# B&R Automation Studio project NAEUL004C00R13L518F00 (part 63)

#### InputRef_Link.var - Change By Project
```iecst
(*2019-06-28*)
(**)
VAR
	p_bLinkStartupRun : REFERENCE TO BOOL;
	p_eLinkMcParamUSCommMod : REFERENCE TO eMcSetCommMod;
	p_bLinkNtParamProjLaneBPrep : REFERENCE TO BOOL;
	bHermesRun : BOOL;
	bHermesStop : BOOL;
END_VAR
(**)
VAR
	p_bLinkDILeftSen : REFERENCE TO BOOL;
	p_eLinkTravLifULPosGo : REFERENCE TO eTravLifULPos;
	p_bLinkOpsTravLifULUSComm : REFERENCE TO BOOL;
END_VAR
(**)
VAR
	sWidthInUMTemp : STRING[80];
END_VAR
```

#### Act_LinkAction.st - Change By Project
```iecst
(** 2021-08-01 **)
ACTION Act_LinkAction:

	IF p_bLinkStartupRun = TRUE THEN
		p_eAct ACCESS p_StartupUSHermesBAct;
	ELSE
		p_eAct ACCESS ADR(eAct);

		IF EDGEPOS(p_eLinkMcParamUSCommMod = McSetCommModHermes AND p_bLinkNtParamProjLaneBPrep) THEN
			bHermesRun	:= TRUE;
			bHermesStop	:= FALSE;
		END_IF

		IF EDGENEG(p_eLinkMcParamUSCommMod = McSetCommModHermes AND p_bLinkNtParamProjLaneBPrep) THEN
			bHermesRun	:= FALSE;
			bHermesStop	:= TRUE;
		END_IF

		IF bHermesRun = TRUE THEN
			p_eAct	:= HermesActBGStartRun;

			IF (eStat = HermesActBGStartRun) AND (eStatus = Done) THEN
				p_eAct		:= HermesActIdle;
				bHermesRun	:= FALSE;
			END_IF
		END_IF

		IF bHermesStop = TRUE THEN
			p_eAct	:= HermesActBGStopRun;

			IF (eStat = HermesActBGStopRun) AND (eStatus = Done) THEN
				p_eAct		:= HermesActIdle;
				bHermesStop	:= FALSE;
			END_IF
		END_IF

		fbDlyTmr(IN := TRUE);
		IF fbDlyTmr.Q THEN
			fbDeleteLogTmr (IN := TRUE);
			IF fbDeleteLogTmr.Q AND eStatus <> Busy THEN
				p_eAct := HermesActDeleteOldLog;
				IF eStat = HermesActDeleteOldLog AND eStatus = Done THEN
					p_eAct := HermesActIdle;
					fbDlyTmr (IN := FALSE);
					fbDeleteLogTmr (IN := FALSE);
				END_IF
			END_IF
		END_IF

	END_IF

END_ACTION
```

#### Act_Link.st - Change By Project
```iecst
(** 2019-06-04 **)
ACTION Act_Link:

	//Receive Alive Time
	p_tyParam.tRcvAlive	:= p_tyParam.tSndAlive * 2;

	//Transfer Complete
	p_bRcvCompl	:= EDGENEG(p_bLinkDILeftSen);

	//Ready Receive
	p_bRdyRcv	:= p_bLinkOpsTravLifULUSComm AND p_eLinkTravLifULPosGo = TravLifULPosUS2;

	//Ready Transport
	p_bRdyTransport	:= TRUE;

	//Accept Data Ready
	IF bUSRdy AND p_eLinkTravLifULPosGo = TravLifULPosUS2 THEN
		p_bAccDataRdy	:= TRUE;
	ELSIF bUSRdy = FALSE THEN
		p_bAccDataRdy	:= FALSE;
	END_IF

	//Accept New Recipe Condition
	p_bAccNewRcpCond	:= p_bOpsRun = TRUE;

	//Info Message
	p_sInfoMsg		:= 'Upstream Hermes Request New Recipe';
	p_sInfoMsg		:= CONCAT(p_sInfoMsg , '$r$n');
	p_sInfoMsg		:= CONCAT(p_sInfoMsg , 'Old Recipe Name : ');
	p_sInfoMsg		:= CONCAT(p_sInfoMsg , p_sRecipeNm);
	p_sInfoMsg		:= CONCAT(p_sInfoMsg , '$r$n');
	p_sInfoMsg		:= CONCAT(p_sInfoMsg , 'Old Recipe Width : ');
	sWidthInUMTemp	:= DINT_TO_STRING(p_diWidthInUM / 1000);
	p_sInfoMsg		:= CONCAT(p_sInfoMsg , sWidthInUMTemp);
	p_sInfoMsg		:= CONCAT(p_sInfoMsg , '$r$n');
	p_sInfoMsg		:= CONCAT(p_sInfoMsg , 'New Recipe Name : ');
	p_sInfoMsg		:= CONCAT(p_sInfoMsg , sReqRecipeNm);
	p_sInfoMsg		:= CONCAT(p_sInfoMsg , '$r$n');
	p_sInfoMsg		:= CONCAT(p_sInfoMsg , 'New Recipe Width : ');
	sWidthInUMTemp	:= DINT_TO_STRING(diReqWidthInUM / 1000);
	p_sInfoMsg		:= CONCAT(p_sInfoMsg , sWidthInUMTemp);

	//Info Message 1 for "SendBoardInfo"
	p_sInfoMsg1     := 'Board Info Received From Upstream';
	p_sInfoMsg1		:= CONCAT(p_sInfoMsg1 , '$r$n');
	p_sInfoMsg1		:= CONCAT(p_sInfoMsg1 , 'PCB Transfer to Last Zone is Blocked');
	p_sInfoMsg1		:= CONCAT(p_sInfoMsg1 , '$r$n');
	p_sInfoMsg1		:= CONCAT(p_sInfoMsg1 , 'Please Insert PCB to Last Zone Outlet');
	p_sInfoMsg1		:= CONCAT(p_sInfoMsg1 , '$r$n');
	p_sInfoMsg1		:= CONCAT(p_sInfoMsg1 , 'and PCB Data Will Be Overwritten');
	p_sInfoMsg1		:= CONCAT(p_sInfoMsg1 , '$r$n');
	p_sInfoMsg1		:= CONCAT(p_sInfoMsg1 , 'To Cancel,unpress the Query Board Info Button');

	//Info Message 2 for "SendBoardInfo"
	p_sInfoMsg2     := 'Board Info Not Found From Upstream';

	//Block Upstream
	//ADD
	//Changed
	bBlkUS :=  bBABlkUS OR bBFBlkUS OR bManuallInsertLastZone; // OR (p_eLinkMcParamUSCommMod = McSetCommModHermes AND (p_bQueryBypassWorkOrder OR p_bNewIncomingBoard)) ; //Remove bManuallInsertLastZone if this is a multiple zones, use bManuallInsertLastZone to block respective zones board transfer

	//Changed
	//For first machine ?
//	IF p_bNewIncomingBoard = FALSE THEN
//		fbUSBlkTm(IN := TRUE);
//	ELSIF p_bNewIncomingBoard THEN
//		fbUSBlkTm(IN := FALSE);
//	END_IF

	//IF AutoRcp Prep, Link
	IF p_bNtParamAutoRcpPrep AND NOT(p_bMcParamAutoRcpDis) AND p_eNtParamAutoRcpPrecededBy = PrecededBySelf   THEN
		p_sRecipeNm	ACCESS p_AutoRcpCurrRcpProdID;
		p_diWidthInUM ACCESS p_AutoRcpCurrRcpWidth;
	ELSE
		p_sRecipeNm	ACCESS p_ProdRcpCurrRcp0Nm;
		p_diWidthInUM ACCESS p_ProdRcpCurrRcp0Width;
	END_IF

END_ACTION
```

#### Cyclic.st - Do Not Change!!!
```iecst
(** 2021-08-01 **)
PROGRAM _CYCLIC

	IF bInitDone = FALSE THEN
		bInitDone	:= TRUE;

		Act_InitLocal;
		Act_InitGlobal;

	ELSIF bInitialDone = FALSE THEN
		IF p_bNtSettingsLoadDone = TRUE THEN
			bInitialDone	:= TRUE;

			Act_Initial;
		END_IF

	ELSE

		Act_RstErr;
		Act_LinkAction;
		Act_Action;
		Act_LinkEn;

		IF (p_bPrep = TRUE) AND (p_bEn = TRUE) AND (p_bDis = FALSE) THEN
			Act_Link;
			Act_Main;
			Act_Background;
			Act_Background_ProcessData;
		ELSE
			Act_Main_Disable;

			IF eStat <> HermesActIdle THEN
				eStatus	:= Done;
			ELSE
				eStatus	:= Idle;
			END_IF
		END_IF

		Act_CombineErr;
		Act_Alarm;
		Act_Alarm1;
		Act_Alarm2;
		Act_Alarm3;
		Act_Alarm4;
		Act_Alarm5;
	END_IF

END_PROGRAM
```

#### Act_InitLocal.st - Do Not Change!!!
```iecst
(** 2021-08-01 **)
ACTION Act_InitLocal:

	//Input Reference Link To Local Variable
	p_eAct ACCESS ADR(eAct);
	p_udiRstErr ACCESS ADR(udiRstErr);
	p_bPrep ACCESS ADR(bPrep);
	p_bEn ACCESS ADR(bEn);
	p_bDis ACCESS ADR(bDis);
	p_tyParam ACCESS ADR(tyParam);
	p_sIPAddr ACCESS ADR(sIPAddr);
	p_tyDTStructure ACCESS ADR(tyDTStructure);
	p_dtCurrDT ACCESS ADR(dtCurrDT);
	p_bRdyRcv ACCESS ADR(bRdyRcv);
	p_bRdyTransport ACCESS ADR(bRdyTransport);
	p_bRcvCompl ACCESS ADR(bRcvCompl);
	p_bRcvIncompl ACCESS ADR(bRcvInCompl);
	p_bRcvNotStart ACCESS ADR(bRcvNotStart);
	p_bBAWidthEn ACCESS ADR(bBAWidthEn);
	p_bBASltEn ACCESS ADR(bBASltEn);
	p_bBFWidthEn ACCESS ADR(bBFWidthEn);
	p_bBFSltEn ACCESS ADR(bBFSltEn);
	p_sMcId ACCESS ADR(sMcId);
	p_sInterfaceId ACCESS ADR(sInterfaceId);
	p_sVersion ACCESS ADR(sVersion);
	p_eFailedBoard ACCESS ADR(eFailedBoard);
	p_sRecipeNm ACCESS ADR(sRecipeNm);
	p_diWidthInUM ACCESS ADR(diWidthInUM);
	p_diMinSltValue ACCESS ADR(diMinSltValue);
	p_diMaxSltValue ACCESS ADR(diMaxSltValue);
	p_diPitch ACCESS ADR(diPitch);
	p_diTtlSlt ACCESS ADR(diTtlSlt);
	p_diSltToSltInUM ACCESS ADR(diSltToSltInUM);
	p_udiSndBffrSize ACCESS ADR(udiSndBffrSize);
	p_udiRcvBffrSize ACCESS ADR(udiRcvBffrSize);
	p_udiAliveIdleTimeInSec ACCESS ADR(udiAliveIdleTimeInSec);
	p_tConnTimeOut ACCESS ADR(tConnTimeOut);
	p_diTransferInTO ACCESS ADR(diTransferInTO);
	p_bOpsRun ACCESS ADR(bOpsRun);
	p_bInterruptSen ACCESS ADR(bInterruptSen);
	p_udiFileKeepDay ACCESS ADR(udiFileKeepDay);
	p_sProgNm ACCESS ADR(sProgNm);
	p_bNtSettingsLoadDone ACCESS ADR(bNtSettingsLoadDone);
	p_bAccDataRdy ACCESS ADR(bAccDataRdy);
	p_bRmtPrep ACCESS ADR(bRmtPrep);
	p_bRmtEn ACCESS ADR(bRmtEn);
	p_bSvyPrep ACCESS ADR(bSvyPrep);
	p_bSvyEn ACCESS ADR(bSvyEn);
	pa_tyProdRcpList ACCESS ADR(a_tyProdRcpList);
	p_tyProdRcpCurrRcp ACCESS ADR(tyProdRcpCurrRcp);
	p_bMcParamMnlAccData ACCESS ADR(bMcParamMnlAccData);
	p_bOpsGConv1HvBrd ACCESS ADR(bOpsGConv1HvBrd);
	p_bManualInsertEndSen ACCESS ADR(bManualInsertEndSen);
	p_bManualInsertZoneHvBrd ACCESS ADR(bManualInsertZoneHvBrd);
	p_bUIAccData ACCESS ADR(bUIAccData);
    p_bQueryBoardInfo ACCESS ADR(bQueryBoardInfo);
	p_sTopBarcode ACCESS ADR(sTopBarcode);
	p_sBottomBarcode ACCESS ADR(sBottomBarcode);
	p_tyHermesConfiguration ACCESS ADR(tyHermesCurrConfiguration);
	p_bTransportFinished ACCESS ADR(bTransportFinished);
	p_bInternalUse ACCESS ADR(bInternalUse);
	p_sInternalRcv ACCESS ADR(sInternalRcv);
	p_bAccNewRcpCond ACCESS ADR(bAccNewRcpCond);
	p_sInfoMsg ACCESS ADR(sInfoMsg);
	p_sInfoMsg1 ACCESS ADR(sInfoMsg1);
	p_sInfoMsg2 ACCESS ADR(sInfoMsg2);

END_ACTION
```

#### Act_Initial.st - Do Not Change!!!
```iecst
(** 2021-08-01 **)
ACTION Act_Initial:

	//Initial
	sStatTxt	:= a_sStatText[eStat];

	fbClntConnect.udiSndBffrSize		:= p_udiSndBffrSize;
	fbClntConnect.udiRcvBffrSize		:= p_udiRcvBffrSize;
	fbClntConnect.udiAliveIdleTmInSec	:= p_udiAliveIdleTimeInSec;
	fbClntConnect.tConnectTO			:= p_tConnTimeOut;
	fbClntConnect(bEn := FALSE);

	fbRcv.udiBffrSize	:= SIZEOF(sRcv);
	fbRcv.p_BffrDest	:= ADR(sRcv);
	fbRcv(bEn := FALSE);

	fbSend.p_BffrDest	:= ADR(sSnd);
	fbSend(bEn := FALSE);

	fbClose(bEn := FALSE);

	fbParseXMLTable.p_XMLTable	:= ADR(a_tyXMLTableDataRcv);

	fbCheckAlive(bEn := FALSE);

	fbCheckAliveSendPing(bEn := FALSE);

	fbCheckAliveRcvPing(bEn := FALSE);

	fbSequenceUS.p_tyMsgTypeRcv	:= ADR(tyMsgTypeRcv);
	fbSequenceUS(bEn := FALSE);

	fbSequenceTO(bEn := FALSE);

	fbFileAppend1.sDevice	:= 'Log';
	fbFileAppend1(bEn := FALSE);

	fbFileOldDel1.sDevice			:= 'Log';
	fbFileOldDel1.sPath				:= '';
	fbFileOldDel1.sKeyword			:= p_sProgNm;
	fbFileOldDel1.udiFileKeepDay	:= p_udiFileKeepDay;
	fbFileOldDel1(bEn := FALSE);

END_ACTION
```

#### Act_Background.st - Do Not Change!!!
```iecst
(** 2021-08-01 **)
ACTION Act_Background:

	IF bRun = TRUE THEN
		IF udiTCPIdent = 0 THEN
			IF p_bInternalUse = FALSE THEN
				Act_Background_TCPConnect;

				tyParamOld	:= p_tyParam;
			ELSE
				udiTCPIdent	:= 1;
			END_IF

		ELSE
			IF bRstConnection = FALSE THEN
				Act_Background_TCPRcv;

				Act_Background_NotificationRcv;
				Act_Background_IllegalMsg;
				Act_Background_ChkParamRcv;
				Act_Background_CmpParamRcv;

				IF bHandshakeDone = TRUE THEN
					IF (p_tyParam.tSndAlive <> T#0s) AND (p_tyParam.tRcvAlive <> T#0s) THEN
						IF tyServiceDescriptionRcv.tyData.tySupportedFeatures.bFeatureCheckAliveResponse = TRUE AND p_tyParam.bFeatureCheckAliveResponse = TRUE THEN
							Act_Background_ChkAliveSendPing;
							Act_Background_ChkAliveRcvPing;
						ELSE
							Act_Background_ChkAlive;
						END_IF
					ELSE
						fbCheckAlive(bEn := FALSE);
						fbCheckAliveSendPing(bEn := FALSE);
						fbCheckAliveRcvPing(bEn := FALSE);
					END_IF
				END_IF

				Act_Background_BoardAvailableChk;
				Act_Background_BoardForecastIdChk;
				Act_Background_Sequence;
				Act_Background_SequenceTO;
				Act_Background_Err;

				IF tyServiceDescriptionRcv.tyAvl.tySupportedFeatures.bFeatureSendBoardInfo = TRUE AND p_tyParam.bFeatureQueryBoardInfo AND bHandshakeDone THEN
					Act_Background_QueryBoardInfo;
				END_IF

				Act_Background_ChgConfig;

				Act_Background_TCPSend;

			//	Act_Background_Log;

			ELSE
				Act_Background_TCPClose;

			END_IF

		END_IF

	    Act_Background_Stop;

	END_IF
	Act_Background_Log;

	IF EDGENEG(bRun) OR EDGENEG(udiTCPIdent = 0) THEN
		//Reset
		fbClntConnect(bEn := FALSE);

		bConnected	:= bRun;
	END_IF

	IF EDGENEG(bRun) OR EDGENEG(udiTCPIdent <> 0) THEN
		fbRcv(bEn := FALSE);
		fbSequenceUS(bEn := FALSE);
		fbSequenceTO(bEn := FALSE);
		fbCheckAlive(bEn := FALSE);
		fbCheckAliveSendPing(bEn := FALSE);
		fbCheckAliveRcvPing(bEn := FALSE);
		fbSend(bEn := FALSE);
		fbClose(bEn := FALSE);

//		fbFileAppend1(bEn := FALSE);
//		iWriteLogStep	:= 0;

		bConnected		    := FALSE;
		bHandshakeDone	    := FALSE;
		bBlkUS			    := FALSE;
		bBABlkUS			:= FALSE;
		bBFBlkUS			:= FALSE;
		bManuallInsertLastZone	:= FALSE;
		bAccDataReq		    := FALSE;
		bBFAccDataReq	    := FALSE;
		bOverWriteSlt    	:= FALSE;
		bOverWriteWidth	    := FALSE;
		bBFOverWriteSlt	    := FALSE;
		bBFOverWriteWidth	:= FALSE;
		bRstConnection    	:= FALSE;
		bRstState	    	:= FALSE;
		bUSRdy	    		:= FALSE;
		bDSRdy		    	:= FALSE;
		bTransporting    	:= FALSE;
		bStopTransport   	:= FALSE;
//		bBAAccpt			:= FALSE;
//		bBFAccpt 			:= FALSE;

		memset(ADR(tyMsgTypeRcv) , 0 , SIZEOF(tyMsgTypeRcv));
		memset(ADR(a_eMsgSend) , 0 , SIZEOF(a_eMsgSend));
		udiMsgSendBffr	:= 0;
	END_IF

	//Reset Error
	IF (eStatus1 = Error) AND bRstErr THEN
		eStatus1	:= Idle;
		udiStatus1	:= 0;

		fbClntConnect(bEn := FALSE);
		fbRcv(bEn := FALSE);
		fbSequenceUS(bEn := FALSE);
		fbSend(bEn := FALSE);
		fbClose(bEn := FALSE);
		fbCheckAlive(bEn := FALSE);
		fbCheckAliveSendPing(bEn := FALSE);
		fbCheckAliveRcvPing(bEn := FALSE);
		fbSequenceTO(bEn := FALSE);

//		fbFileAppend1(bEn := FALSE);
//		iWriteLogStep	:= 0;

		bConnected		    := FALSE;
		bHandshakeDone	    := FALSE;
		bBlkUS			    := FALSE;
		bBABlkUS			:= FALSE;
		bBFBlkUS			:= FALSE;
		bManuallInsertLastZone	:= FALSE;
		bAccDataReq		    := FALSE;
		bBFAccDataReq	    := FALSE;
		bOverWriteSlt    	:= FALSE;
		bOverWriteWidth	    := FALSE;
		bBFOverWriteSlt	    := FALSE;
		bBFOverWriteWidth	:= FALSE;
		bRstConnection    	:= FALSE;
		bRstState	    	:= FALSE;
		bUSRdy	    		:= FALSE;
		bDSRdy		    	:= FALSE;
		bTransporting    	:= FALSE;
		bStopTransport   	:= FALSE;

		memset(ADR(tyMsgTypeRcv) , 0 , SIZEOF(tyMsgTypeRcv));
		memset(ADR(a_eMsgSend) , 0 , SIZEOF(a_eMsgSend));
		udiMsgSendBffr	:= 0;
	END_IF

	IF (eStatus2 = Error) AND bRstErr THEN
		eStatus2	:= Idle;
		udiStatus2	:= 0;

		fbSequenceTO(bEn := FALSE);

	END_IF

	IF (eStatus3 = Error) AND bRstErr THEN
		eStatus3	:= Idle;
		udiStatus3	:= 0;

//		fbFileAppend1(bEn := FALSE);
//		iWriteLogStep	:= 0;
	END_IF

	IF (eStatus4 = Error) AND bRstErr THEN
		eStatus4	:= Idle;
		udiStatus4	:= 0;
	END_IF

	Act_Background_AccData;
	Act_Background_BFAccData;

END_ACTION
```

#### Act_Background_ProcessData.st - Do Not Change!!!
```iecst
(** 2021-08-01 **)
ACTION Act_Background_ProcessData:

    //Pass Board Available data and bStopTransportSnd BOOL to "BoardArrived" (SupervisoryHermes)
	IF EDGEPOS (fbSequenceUS.eMsgTypeSnd = HermesMsgTypeStopTransport) AND p_bOpsGConv1HvBrd THEN //Incoming Zone have board
		tyBoardArrivedInfo := tyBoardAvailableRcv;
		bStopTransportSnd := TRUE;
	END_IF

	//Auto Reset bStopTransportSnd
	fbSendTm(IN := bStopTransportSnd, PT := T#0.5S);
	IF fbSendTm.Q = TRUE THEN
		fbSendTm(IN := FALSE);
		bStopTransportSnd	:= FALSE;
	END_IF

	//Process BoardForecast(Id) or BoardForecast()
	bFeatureBoardForecast := (p_tyParam.bFeatureBoardForecast = TRUE) AND (tyServiceDescriptionRcv.tyAvl.tySupportedFeatures.bFeatureBoardForecast = TRUE);

	IF bFeatureBoardForecast THEN
		IF tyMsgTypeRcv.bBoardForecast AND tyBoardForecastRcv.tyData.sForecastId <> '' AND bProcessBoardForecastId = FALSE AND fbDelayTm.Q AND bBFAccDataReq = FALSE AND bManuallInsertLastZone = FALSE THEN
			bProcessBoardForecastId := TRUE; //Process BoardForecast(Id)
			tyBoardForecastAcc := tyBoardForecastRcv;
			tyMsgTypeRcv.bBoardForecast := FALSE;
			fbDelayTm(IN := FALSE);
		ELSIF tyMsgTypeRcv.bBoardForecast AND tyBoardForecastRcv.tyData.sForecastId = '' AND bProcessBoardForecastId = FALSE THEN //Process BoardForecast()
			tyBoardForecastAcc := tyBoardForecastRcv;
			tyMsgTypeRcv.bBoardForecast := FALSE;
		END_IF
	ELSE
		bProcessBoardForecastId := FALSE;
	END_IF

	//Next PCB incoming time
	tNextPCBTm := REAL_TO_TIME((tyBoardForecastAcc.tyData.rTimeUntilAvailable)*1000);

    //Delay 0.5s to process another new BoardForecast(Id)
	fbDelayTm(IN := NOT bProcessBoardForecastId, PT := T#0.5S);

	//Ready Transport
	p_bRdyTransport	:= bRdyTransport;

	//Auto Reset bStopTransportSnd
	fbCheckBATimer(IN := bBoardAvailable AND (fbSequenceUS.eState = HermesStateAvailableAndReady) AND (bBlkUS = FALSE), PT := T#0.1S); //need this small delay to compare recipe & width, before board transfer can happens
	IF fbCheckBATimer.Q = TRUE THEN
		fbCheckBATimer(IN := FALSE);
		bRdyTransport := TRUE;
	ELSE
		bRdyTransport := FALSE;
	END_IF

END_ACTION
```

#### Act_Background_TCPConnect.st - Do Not Change!!!
```iecst
(** 2021-08-01 **)
ACTION Act_Background_TCPConnect:

	IF eStatus1 <> Error AND eStatus2 <> Error THEN

		//Connect Server
		fbClntConnect.sClntIP		:= p_sIPAddr;
		fbClntConnect.sSvrIP		:= p_tyParam.sHostAddress;
		fbClntConnect.uiClntPort	:= p_tyParam.uiClntPort;
		fbClntConnect.uiSvrPort		:= p_tyParam.uiHostPort;
		fbClntConnect(bEn := TRUE);

		IF fbClntConnect.udiStatus = 0 THEN
			udiTCPIdent	:= fbClntConnect.udiTCPIdent;
			fbClntConnect(bEn := FALSE);

		ELSIF fbClntConnect.udiStatus = 2313 THEN
			fbClntConnect(bEn := FALSE);

		ELSIF fbClntConnect.udiStatus = 2323 OR bConnected= FALSE THEN
			udiStatus5	:= 10013;	//US Hermes Connection Lost

		ELSIF fbClntConnect.udiStatus < 65534 THEN
			eStatus1	:= Error;

			IF fbClntConnect.udiStatus = 2300 THEN
				udiStatus1	:= 10000;	//Invalid Ident While Client Connecting
			ELSIF fbClntConnect.udiStatus = 2302 THEN
				udiStatus1	:= 10001;	//Setting Keep Alive Interval Time Error While Client Connecting
			ELSIF fbClntConnect.udiStatus = 2303 THEN
				udiStatus1	:= 10002;	//Setting Keep Alive Idle Time Error While Client Connecting
			ELSIF fbClntConnect.udiStatus = 2304 THEN
				udiStatus1	:= 10003;	//Setting Keep Alive Count Error While Client Connecting
			ELSIF fbClntConnect.udiStatus = 2305 THEN
				udiStatus1	:= 10004;	//Setting Keep Alive Error While Client Connecting
			ELSIF fbClntConnect.udiStatus = 2306 THEN
				udiStatus1	:= 10005;	//Setting Receive Buffer Error While Client Connecting
			ELSIF fbClntConnect.udiStatus = 2307 THEN
				udiStatus1	:= 10006;	//Setting Send Buffer Error While Client Connecting
			ELSIF fbClntConnect.udiStatus = 2308 THEN
				udiStatus1	:= 10007;	//Setting No Waiting Error While Client Connecting
			ELSIF fbClntConnect.udiStatus = 2309 THEN
				udiStatus1	:= 10008;	//TCP Open Port Error While Client Connecting
			ELSIF fbClntConnect.udiStatus = 2310 THEN
				udiStatus1	:= 10009;	//Closing TCP Error While Client Connecting
			ELSIF fbClntConnect.udiStatus = 2313 THEN
				udiStatus1	:= 10010;	//Server Connection Failed While Client Connecting
			ELSIF fbClntConnect.udiStatus = 2314 THEN
				udiStatus1	:= 10011;	//Ident In Used While Client Connecting
			ELSIF fbClntConnect.udiStatus = 2315 THEN
				udiStatus1	:= 10012;	//Connect To Server Error While Client Connecting
			ELSE
				udiStatus1	:= fbClntConnect.udiStatus;
			END_IF

		END_IF

	END_IF

END_ACTION
```

#### Act_Background_TCPRcv.st - Do Not Change!!!
```iecst
(** 2021-08-01 **)
ACTION Act_Background_TCPRcv:

	IF eStatus1 <> Error THEN

		//Receive Data
		IF p_bInternalUse = FALSE THEN
			fbRcv.udiTCPIdent	:= udiTCPIdent;
			fbRcv(bEn := TRUE);
		ELSE
			sRcv	:= p_sInternalRcv;
		END_IF

		IF (fbRcv.udiStatus = 0) OR ((p_bInternalUse = TRUE) AND (LEN(sRcv) > 0)) THEN

			fLogDTConvert(ADR(sDT) , p_dtCurrDT);
			memset(ADR(a_sLogList[udiLogCntr]) , 0 , SIZEOF(a_sLogList[udiLogCntr]));
			memcpy(ADR(a_sLogList[udiLogCntr]) + LEN(a_sLogList[udiLogCntr]) , ADR(sDT) , LEN(sDT));
			memcpy(ADR(a_sLogList[udiLogCntr]) + LEN(a_sLogList[udiLogCntr]) , ADR('$r$n') , LEN('$r$n'));
			memcpy(ADR(a_sLogList[udiLogCntr]) + LEN(a_sLogList[udiLogCntr]) , ADR('RCV_FRM_US$r$n') , LEN('RCV_FRM_US$r$n'));
			memcpy(ADR(a_sLogList[udiLogCntr]) + LEN(a_sLogList[udiLogCntr]) , ADR(sRcv) , LEN(sRcv));
			memcpy(ADR(a_sLogList[udiLogCntr]) + LEN(a_sLogList[udiLogCntr]) , ADR('$r$n$r$n') , LEN('$r$n$r$n'));

			udiLogCntr	:= udiLogCntr + 1;
			IF udiLogCntr = 11 THEN
				udiLogCntr	:= 1;
			END_IF

			fXMLConvertToTable(ADR(sRcv) , LEN(sRcv) , ADR(a_tyXMLTableDataRcv) , ADR(a_tyXMLTableDataRcv[0].sTitle) , SIZEOF(a_tyXMLTableDataRcv[0].sTitle) , ADR(a_tyXMLTableDataRcv[0].sValue) , SIZEOF(a_tyXMLTableDataRcv[0].sValue) , ADR(a_tyXMLTableDataRcv[0].uiSize) , SIZEOF(a_tyXMLTableDataRcv[0]) , SIZEOF(a_tyXMLTableDataRcv) / SIZEOF(a_tyXMLTableDataRcv[0]) , ADR(udiXMLTableWriteIdx));

			fbParseXMLTable.iTotalIdxWrite	:= UDINT_TO_INT(udiXMLTableWriteIdx);
			fbParseXMLTable;

			IF fbParseXMLTable.tyMsgType.bCheckAlive = TRUE THEN
				tyMsgTypeRcv.bCheckAlive	:= TRUE;
				tyCheckAliveRcv				:= fbParseXMLTable.tyCheckAlive;
			END_IF

			IF fbParseXMLTable.tyMsgType.bCheckAlivePing = TRUE THEN
				tyMsgTypeRcv.bCheckAlivePing	:= TRUE;
				tyCheckAlivePingRcv				:= fbParseXMLTable.tyCheckAlivePing;
			END_IF

			IF fbParseXMLTable.tyMsgType.bCheckAlivePong = TRUE THEN
				tyMsgTypeRcv.bCheckAlivePong	:= TRUE;
				tyCheckAlivePongRcv				:= fbParseXMLTable.tyCheckAlivePong;
			END_IF

			IF fbParseXMLTable.tyMsgType.bServiceDescription = TRUE THEN
				tyMsgTypeRcv.bServiceDescription	:= TRUE;
				tyServiceDescriptionRcv				:= fbParseXMLTable.tyServiceDescription;
			END_IF

			IF fbParseXMLTable.tyMsgType.bNotification = TRUE THEN
				tyMsgTypeRcv.bNotification	:= TRUE;
				tyNotificationRcv			:= fbParseXMLTable.tyNotification;
			END_IF

			IF fbParseXMLTable.tyMsgType.bBoardAvailable = TRUE THEN
				tyMsgTypeRcv.bBoardAvailable	:= TRUE;
				tyBoardAvailableRcv				:= fbParseXMLTable.tyBoardAvailable;

				memset(ADR(a_tyXMLTableDataBrdAvl) , 0 , SIZEOF(a_tyXMLTableDataBrdAvl));
				memcpy(ADR(a_tyXMLTableDataBrdAvl) , ADR(a_tyXMLTableDataRcv) + (fbParseXMLTable.iBoardAvailableFirstIdx * SIZEOF(a_tyXMLTableDataRcv[0])) , (fbParseXMLTable.iBoardAvailableLastIdx - fbParseXMLTable.iBoardAvailableFirstIdx + 1) * SIZEOF(a_tyXMLTableDataRcv[0]));

				iXMLTableDataBrdAvlTtlIdx	:= fbParseXMLTable.iBoardAvailableLastIdx - fbParseXMLTable.iBoardAvailableFirstIdx + 1;

			END_IF

			IF fbParseXMLTable.tyMsgType.bRevokeBoardAvailable = TRUE THEN
				tyMsgTypeRcv.bRevokeBoardAvailable	:= TRUE;
			END_IF

			IF fbParseXMLTable.tyMsgType.bMachineReady = TRUE THEN
				tyMsgTypeRcv.bMachineReady	:= TRUE;
				tyMachineReady				:= fbParseXMLTable.tyMachineReady;
			END_IF

			IF fbParseXMLTable.tyMsgType.bRevokeMachineReady = TRUE THEN
				tyMsgTypeRcv.bRevokeMachineReady	:= TRUE;
			END_IF

			IF fbParseXMLTable.tyMsgType.bStartTransport = TRUE THEN
				tyMsgTypeRcv.bStartTransport	:= TRUE;
				tyStartTransport				:= fbParseXMLTable.tyStartTransport;
			END_IF

			IF fbParseXMLTable.tyMsgType.bStopTransport = TRUE THEN
				tyMsgTypeRcv.bStopTransport	:= TRUE;
				tyStopTransport				:= fbParseXMLTable.tyStopTransport;
			END_IF

			IF fbParseXMLTable.tyMsgType.bTransportFinished = TRUE THEN
				tyMsgTypeRcv.bTransportFinished	:= TRUE;
				tyTransportFinished				:= fbParseXMLTable.tyTransportFinished;
			END_IF

			IF fbParseXMLTable.tyMsgType.bSetConfiguration = TRUE THEN
				tyMsgTypeRcv.bSetConfiguration	:= TRUE;
				tySetConfiguration				:= fbParseXMLTable.tySetConfiguration;
			END_IF

			IF fbParseXMLTable.tyMsgType.bGetConfiguration = TRUE THEN
				tyMsgTypeRcv.bGetConfiguration	:= TRUE;
			END_IF

			IF fbParseXMLTable.tyMsgType.bCurrentConfiguration = TRUE THEN
				tyMsgTypeRcv.bCurrentConfiguration	:= TRUE;
				tyCurrentConfiguration				:= fbParseXMLTable.tyCurrentConfiguration;
			END_IF

			IF fbParseXMLTable.tyMsgType.bBoardForecast = TRUE THEN
				tyMsgTypeRcv.bBoardForecast	:= TRUE;
				tyBoardForecastRcv				:= fbParseXMLTable.tyBoardForecast;
			END_IF

			IF fbParseXMLTable.tyMsgType.bQueryBoardInfo = TRUE THEN
				tyMsgTypeRcv.bQueryBoardInfo	:= TRUE;
				tyQueryBoardInfo				:= fbParseXMLTable.tyQueryBoardInfo;
			END_IF

			IF fbParseXMLTable.tyMsgType.bSendBoardInfo = TRUE THEN
				tyMsgTypeRcv.bSendBoardInfo	:= TRUE;
				tySendBoardInfoRcv				:= fbParseXMLTable.tySendBoardInfo;
			END_IF

			fbRcv(bEn := FALSE);

			memset(ADR(sRcv) , 0 , SIZEOF(sRcv));

		ELSIF (fbRcv.udiStatus = 2317) AND (p_bInternalUse = FALSE) THEN
			fbRcv(bEn := FALSE);

			memset(ADR(sRcv) , 0 , SIZEOF(sRcv));

		ELSIF (fbRcv.udiStatus = 2316) AND (p_bInternalUse = FALSE) THEN
			bRstConnection	:= TRUE;

			memset(ADR(sRcv) , 0 , SIZEOF(sRcv));

		ELSIF (fbRcv.udiStatus = 2318) AND (p_bInternalUse = FALSE) THEN
			bRstConnection	:= TRUE;

			memset(ADR(sRcv) , 0 , SIZEOF(sRcv));

		ELSIF (fbRcv.udiStatus < 65534) AND (p_bInternalUse = FALSE) THEN
			eStatus1	:= Error;

			IF fbRcv.udiStatus = 2300 THEN
				udiStatus1	:= 10014;	//Invalid Ident While Receiving Data
			ELSIF fbRcv.udiStatus = 2319 THEN
				udiStatus1	:= 10015;	//TCP Receive Data Error While Receiving Data
			ELSE
				udiStatus1	:= fbRcv.udiStatus;
			END_IF

			memset(ADR(sRcv) , 0 , SIZEOF(sRcv));

		END_IF

	END_IF

END_ACTION
```

#### Act_Background_IllegalMsg.st - Do Not Change!!!
```iecst
(** 2021-08-01 **)
ACTION Act_Background_IllegalMsg:

	IF eStatus2 <> Error THEN

		udiStatus2	:= fHermesIllegalMsgUS(fbSequenceUS.eState , tyMsgTypeRcv , fbSequenceUS.bBoardAvailable);

		IF udiStatus2 <> 0 THEN
			eStatus2	:= Error;

			IF udiStatus2 = 2770 THEN
				udiStatus2	:= 10016;	//Receive ServiceDescription While Upstream In Not Connected State
			ELSIF udiStatus2 = 2771 THEN
				udiStatus2	:= 10017;	//Receive BoardAvailable While Upstream In Not Connected State
			ELSIF udiStatus2 = 2772 THEN
				udiStatus2	:= 10018;	//Receive RevokeBoardAvailable While Upstream In Not Connected State
			ELSIF udiStatus2 = 2773 THEN
				udiStatus2	:= 10019;	//Receive MachineReady While Upstream In Not Connected State
			ELSIF udiStatus2 = 2774 THEN
				udiStatus2	:= 10020;	//Receive RevokeMachineReady While Upstream In Not Connected State
			ELSIF udiStatus2 = 2775 THEN
				udiStatus2	:= 10021;	//Receive StartTransport While Upstream In Not Connected State
			ELSIF udiStatus2 = 2776 THEN
				udiStatus2	:= 10022;	//Receive StopTransport While Upstream In Not Connected State
			ELSIF udiStatus2 = 2777 THEN
				udiStatus2	:= 10023;	//Receive TransportFinished While Upstream In Not Connected State
			ELSIF udiStatus2 = 2778 THEN
				udiStatus2	:= 10024;	//Receive BoardForecast While Upstream In Not Connected State
			ELSIF udiStatus2 = 2779 THEN
				udiStatus2	:= 10025;	//Receive BoardAvailable While Upstream In Service Description State
			ELSIF udiStatus2 = 2780 THEN
				udiStatus2	:= 10026;	//Receive RevokeBoardAvailable While Upstream In Service Description State
			ELSIF udiStatus2 = 2781 THEN
				udiStatus2	:= 10027;	//Receive MachineReady While Upstream In Service Description State
			ELSIF udiStatus2 = 2782 THEN
				udiStatus2	:= 10028;	//Receive RevokeMachineReady While Upstream In Service Description State
			ELSIF udiStatus2 = 2783 THEN
				udiStatus2	:= 10029;	//Receive StartTransport While Upstream In Service Description State
			ELSIF udiStatus2 = 2784 THEN
				udiStatus2	:= 10030;	//Receive StopTransport While Upstream In Service Description State
			ELSIF udiStatus2 = 2785 THEN
				udiStatus2	:= 10031;	//Receive TransportFinished While Upstream In Service Description State
			ELSIF udiStatus2 = 2786 THEN
				udiStatus2	:= 10032;	//Receive BoardForecast While Upstream In Service Description State
			ELSIF udiStatus2 = 2787 THEN
				udiStatus2	:= 10033;	//Receive ServiceDescription While Upstream In Not Available Not Ready State
			ELSIF udiStatus2 = 2788 THEN
				udiStatus2	:= 10034;	//Receive RevokeBoardAvailable While Upstream In Not Available Not Ready State
			ELSIF udiStatus2 = 2789 THEN
				udiStatus2	:= 10035;	//Receive MachineReady While Upstream In Not Available Not Ready State
			ELSIF udiStatus2 = 2790 THEN
				udiStatus2	:= 10036;	//Receive RevokeMachineReady While Upstream In Not Available Not Ready State
			ELSIF udiStatus2 = 2791 THEN
				udiStatus2	:= 10037;	//Receive StartTransport While Upstream In Not Available Not Ready State
			ELSIF udiStatus2 = 2792 THEN
				udiStatus2	:= 10038;	//Receive StopTransport While Upstream In Not Available Not Ready State
			ELSIF udiStatus2 = 2793 THEN
				udiStatus2	:= 10039;	//Receive TransportFinished While Upstream In Not Available Not Ready State
			ELSIF udiStatus2 = 2794 THEN
				udiStatus2	:= 10040;	//Receive ServiceDescription While Upstream In Board Available State
			ELSIF udiStatus2 = 2795 THEN
				udiStatus2	:= 10041;	//Receive BoardAvailable While Upstream In Board Available State
			ELSIF udiStatus2 = 2796 THEN
				udiStatus2	:= 10042;	//Receive MachineReady While Upstream In Board Available State
			ELSIF udiStatus2 = 2797 THEN
				udiStatus2	:= 10043;	//Receive RevokeMachineReady While Upstream In Board Available State
			ELSIF udiStatus2 = 2798 THEN
				udiStatus2	:= 10044;	//Receive StartTransport While Upstream In Board Available State
			ELSIF udiStatus2 = 2799 THEN
				udiStatus2	:= 10045;	//Receive StopTransport While Upstream In Board Available State
			ELSIF udiStatus2 = 2800 THEN
				udiStatus2	:= 10046;	//Receive TransportFinished While Upstream In Board Available State
			ELSIF udiStatus2 = 2801 THEN
				udiStatus2	:= 10047;	//Receive BoardForecast While Upstream In Board Available State
			ELSIF udiStatus2 = 2802 THEN
				udiStatus2	:= 10048;	//Receive ServiceDescription While Upstream In Machine Ready State
			ELSIF udiStatus2 = 2803 THEN
				udiStatus2	:= 10049;	//Receive RevokeBoardAvailable While Upstream In Machine Ready State
			ELSIF udiStatus2 = 2804 THEN
				udiStatus2	:= 10050;	//Receive MachineReady While Upstream In Machine Ready State
			ELSIF udiStatus2 = 2805 THEN
				udiStatus2	:= 10051;	//Receive RevokeMachineReady While Upstream In Machine Ready State
			ELSIF udiStatus2 = 2806 THEN
				udiStatus2	:= 10052;	//Receive StartTransport While Upstream In Machine Ready State
			ELSIF udiStatus2 = 2807 THEN
				udiStatus2	:= 10053;	//Receive StopTransport While Upstream In Machine Ready State
			ELSIF udiStatus2 = 2808 THEN
				udiStatus2	:= 10054;	//Receive TransportFinished While Upstream In Machine Ready State
			ELSIF udiStatus2 = 2809 THEN
				udiStatus2	:= 10055;	//Receive ServiceDescription While Upstream In Available And Ready State
			ELSIF udiStatus2 = 2810 THEN
				udiStatus2	:= 10056;	//Receive BoardAvailable While Upstream In Available And Ready State
			ELSIF udiStatus2 = 2811 THEN
				udiStatus2	:= 10057;	//Receive MachineReady While Upstream In Available And Ready State
			ELSIF udiStatus2 = 2812 THEN
				udiStatus2	:= 10058;	//Receive RevokeMachineReady While Upstream In Available And Ready State
			ELSIF udiStatus2 = 2813 THEN
				udiStatus2	:= 10059;	//Receive StartTransport While Upstream In Available And Ready State
			ELSIF udiStatus2 = 2814 THEN
				udiStatus2	:= 10060;	//Receive StopTransport While Upstream In Available And Ready State
			ELSIF udiStatus2 = 2815 THEN
				udiStatus2	:= 10061;	//Receive TransportFinished While Upstream In Available And Ready State
			ELSIF udiStatus2 = 2816 THEN
				udiStatus2	:= 10062;	//Receive BoardForecast While Upstream In Available And Ready State
			ELSIF udiStatus2 = 2817 THEN
				udiStatus2	:= 10063;	//Receive ServiceDescription While Upstream In Transporting State
			ELSIF udiStatus2 = 2818 THEN
				udiStatus2	:= 10064;	//Receive Twice Board Available While Upstream In Transporting State
			ELSIF udiStatus2 = 2819 THEN
				udiStatus2	:= 10065;	//Receive RevokeBoardAvailable Without BoardAvailable While Upstream In Transporting State
			ELSIF udiStatus2 = 2820 THEN
				udiStatus2	:= 10066;	//Receive MachineReady While Upstream In Transporting State
			ELSIF udiStatus2 = 2821 THEN
				udiStatus2	:= 10067;	//Receive RevokeMachineReady While Upstream In Transporting State
			ELSIF udiStatus2 = 2822 THEN
				udiStatus2	:= 10068;	//Receive StartTransport While Upstream In Transporting State
			ELSIF udiStatus2 = 2823 THEN
				udiStatus2	:= 10069;	//Receive StopTransport While Upstream In Transporting State
			ELSIF udiStatus2 = 2824 THEN
				udiStatus2	:= 10070;	//Receive ServiceDescription While Upstream In Transport Finished State
			ELSIF udiStatus2 = 2825 THEN
				udiStatus2	:= 10071;	//Receive BoardAvailable While Upstream In Transport Finished State
			ELSIF udiStatus2 = 2826 THEN
				udiStatus2	:= 10072;	//Receive RevokeBoardAvailable While UpstreamWhile Upstream In Transport Finished State
			ELSIF udiStatus2 = 2827 THEN
				udiStatus2	:= 10073;	//Receive MachineReady While Upstream In Transport Finished State
			ELSIF udiStatus2 = 2828 THEN
				udiStatus2	:= 10074;	//Receive RevokeMachineReady While Upstream In Transport Finished State
			ELSIF udiStatus2 = 2829 THEN
				udiStatus2	:= 10075;	//Receive StartTransport While Upstream In Transport Finished State
			ELSIF udiStatus2 = 2830 THEN
				udiStatus2	:= 10076;	//Receive TransportFinished While Upstream In Transport Finished State
			ELSIF udiStatus2 = 2831 THEN
				udiStatus2	:= 10077;	//Receive StopTransport While Upstream In Transport Finished State
			ELSIF udiStatus2 = 2832 THEN
				udiStatus2	:= 10078;	//Receive BoardForecast While Upstream In Transport Finished State
			ELSIF udiStatus2 = 2833 THEN
				udiStatus2	:= 10079;	//Receive ServiceDescription While Upstream In Transport Stopped State
			ELSIF udiStatus2 = 2834 THEN
				udiStatus2	:= 10080;	//Receive Twice Board Available While Upstream In Transport Stopped State
			ELSIF udiStatus2 = 2835 THEN
				udiStatus2	:= 10081;	//Receive RevokeBoardAvailable Without BoardAvailable While Upstream In Transport Stopped State
			ELSIF udiStatus2 = 2836 THEN
				udiStatus2	:= 10082;	//Receive MachineReady While Upstream In Transport Stopped State
			ELSIF udiStatus2 = 2837 THEN
				udiStatus2	:= 10083;	//Receive RevokeMachineReady While Upstream In Transport Stopped State
			ELSIF udiStatus2 = 2838 THEN
				udiStatus2	:= 10084;	//Receive StartTransport While Upstream In Transport Stopped State
			ELSIF udiStatus2 = 2839 THEN
				udiStatus2	:= 10085;	//Receive StopTransport While Upstream In Transport Stopped State
			END_IF

			fHermesAddOneMsgSend(ADR(a_eMsgSend) , ADR(udiMsgSendBffr) , HermesMsgTypeNotification);

			tyNotificationSnd.tyAvl.bSeverity			:= TRUE;
			tyNotificationSnd.tyAvl.bNotificationCode	:= TRUE;
			tyNotificationSnd.tyAvl.bDescription		:= TRUE;
			tyNotificationSnd.tyData.eSeverity			:= HermesSeverityFatalError;
			tyNotificationSnd.tyData.iNotificationCode	:= UDINT_TO_INT(udiStatus2);
			tyNotificationSnd.tyData.sDescription		:= a_tyAlmText[udiStatus2].sAlmText;

		END_IF

	END_IF

END_ACTION
```

#### Act_Background_ChkParamRcv.st - Do Not Change!!!
```iecst
(** 2021-08-01 **)
ACTION Act_Background_ChkParamRcv:

	IF eStatus2 <> Error THEN

		//Check Parameter Receive
		IF tyMsgTypeRcv.bServiceDescription = TRUE THEN
			udiStatus2	:= fHermesChkParamSD(tyServiceDescriptionRcv , p_tyParam.iLaneID);

			IF udiStatus2 = 2731 THEN
				udiStatus2	:= 0;
			END_IF

			IF udiStatus2 <> 0 THEN
				eStatus2	:= Error;

				IF udiStatus2 = 2726 THEN
					udiStatus2	:= 10086;	//LaneId Mismatch While Checking Service Description
				ELSIF udiStatus2 = 2727 THEN
					udiStatus2	:= 10087;	//MachineId Missing While Checking Service Description
				ELSIF udiStatus2 = 2728 THEN
					udiStatus2	:= 10088;	//LandId Out Of Range While Checking Service Description
				ELSIF udiStatus2 = 2729 THEN
					udiStatus2	:= 10089;	//LandId Missing While Checking Service Description
				ELSIF udiStatus2 = 2730 THEN
					udiStatus2	:= 10090;	//Version Missing While Checking Service Description
				ELSIF udiStatus2 = 2731 THEN
					udiStatus2	:= 10091;	//SupportedFeatures Missing While Checking Service Description
				END_IF

				fHermesAddOneMsgSend(ADR(a_eMsgSend) , ADR(udiMsgSendBffr) , HermesMsgTypeNotification);

				tyNotificationSnd.tyAvl.bSeverity			:= TRUE;
				tyNotificationSnd.tyAvl.bNotificationCode	:= TRUE;
				tyNotificationSnd.tyAvl.bDescription		:= TRUE;
				tyNotificationSnd.tyData.eSeverity			:= HermesSeverityFatalError;
				tyNotificationSnd.tyData.iNotificationCode	:= UDINT_TO_INT(udiStatus2);
				tyNotificationSnd.tyData.sDescription		:= a_tyAlmText[udiStatus2].sAlmText;

			END_IF
		END_IF

		IF tyMsgTypeRcv.bNotification = TRUE THEN
			udiStatus2	:= fHermesChkParamN(tyNotificationRcv);

			IF udiStatus2 <> 0 THEN
				eStatus2	:= Error;

				IF udiStatus2 = 2732 THEN
					udiStatus2	:= 10092;	//NotificationCode Out Of Range While Checking Notification
				ELSIF udiStatus2 = 2733 THEN
					udiStatus2	:= 10093;	//NotificationCode Missing While Checking Notification
				ELSIF udiStatus2 = 2734 THEN
					udiStatus2	:= 10094;	//Severity Missing While Checking Notification
				ELSIF udiStatus2 = 2735 THEN
					udiStatus2	:= 10095;	//Description Missing While Checking Notification
				END_IF

				fHermesAddOneMsgSend(ADR(a_eMsgSend) , ADR(udiMsgSendBffr) , HermesMsgTypeNotification);

				tyNotificationSnd.tyAvl.bSeverity			:= TRUE;
				tyNotificationSnd.tyAvl.bNotificationCode	:= TRUE;
				tyNotificationSnd.tyAvl.bDescription		:= TRUE;
				tyNotificationSnd.tyData.eSeverity			:= HermesSeverityFatalError;
				tyNotificationSnd.tyData.iNotificationCode	:= UDINT_TO_INT(udiStatus2);
				tyNotificationSnd.tyData.sDescription		:= a_tyAlmText[udiStatus2].sAlmText;

			END_IF
		END_IF

		IF tyMsgTypeRcv.bBoardAvailable = TRUE THEN
			udiStatus2	:= fHermesChkParamBA(tyBoardAvailableRcv);

			IF udiStatus2 <> 0 THEN
				eStatus2	:= Error;

				IF udiStatus2 = 2736 THEN
					udiStatus2	:= 10096;	//BoardId Missing While Checking Board Available
				ELSIF udiStatus2 = 2737 THEN
					udiStatus2	:= 10097;	//BoardIdCreatedBy Missing While Checking Board Available
				ELSIF udiStatus2 = 2738 THEN
					udiStatus2	:= 10098;	//FailedBoard Missing While Checking Board Available
				ELSIF udiStatus2 = 2739 THEN
					udiStatus2	:= 10099;	//FlippedBoard Missing While Checking Board Available
				END_IF

				fHermesAddOneMsgSend(ADR(a_eMsgSend) , ADR(udiMsgSendBffr) , HermesMsgTypeNotification);

				tyNotificationSnd.tyAvl.bSeverity			:= TRUE;
				tyNotificationSnd.tyAvl.bNotificationCode	:= TRUE;
				tyNotificationSnd.tyAvl.bDescription		:= TRUE;
				tyNotificationSnd.tyData.eSeverity			:= HermesSeverityError;
				tyNotificationSnd.tyData.iNotificationCode	:= UDINT_TO_INT(udiStatus2);
				tyNotificationSnd.tyData.sDescription		:= a_tyAlmText[udiStatus2].sAlmText;

			END_IF

		END_IF

		IF tyMsgTypeRcv.bTransportFinished = TRUE THEN
			udiStatus2	:= fHermesChkParamTF(tyTransportFinished);

			IF udiStatus2 <> 0 THEN
				eStatus2	:= Error;

				IF udiStatus2 = 2744 THEN
					udiStatus2	:= 10100;	//TransferState Missing While Checking Transport Finished
				ELSIF udiStatus2 = 2745 THEN
					udiStatus2	:= 10101;	//BoardId Missing While Checking Transport Finished
				END_IF

				fHermesAddOneMsgSend(ADR(a_eMsgSend) , ADR(udiMsgSendBffr) , HermesMsgTypeNotification);

				tyNotificationSnd.tyAvl.bSeverity			:= TRUE;
				tyNotificationSnd.tyAvl.bNotificationCode	:= TRUE;
				tyNotificationSnd.tyAvl.bDescription		:= TRUE;
				tyNotificationSnd.tyData.eSeverity			:= HermesSeverityError;
				tyNotificationSnd.tyData.iNotificationCode	:= UDINT_TO_INT(udiStatus2);
				tyNotificationSnd.tyData.sDescription		:= a_tyAlmText[udiStatus2].sAlmText;

			END_IF
		END_IF

		IF tyMsgTypeRcv.bBoardForecast = TRUE THEN
			IF bFeatureBoardForecast = TRUE THEN

				udiStatus2	:= fHermesChkParamBF(tyBoardForecastRcv);

				IF udiStatus2 <> 0 THEN
					eStatus2	:= Error;

					IF udiStatus2 = 2764 THEN
						udiStatus2	:= 10102;	//FailedBoard Missing While Checking Board Forecast

					ELSIF udiStatus2 = 2765 THEN
						udiStatus2	:= 10103;	//FlippedBoard Missing While Checking Board Forecast
					END_IF

					fHermesAddOneMsgSend(ADR(a_eMsgSend) , ADR(udiMsgSendBffr) , HermesMsgTypeNotification);

					tyNotificationSnd.tyAvl.bSeverity			:= TRUE;
					tyNotificationSnd.tyAvl.bNotificationCode	:= TRUE;
					tyNotificationSnd.tyAvl.bDescription		:= TRUE;
					tyNotificationSnd.tyData.eSeverity			:= HermesSeverityError;
					tyNotificationSnd.tyData.iNotificationCode	:= UDINT_TO_INT(udiStatus2);
					tyNotificationSnd.tyData.sDescription		:= a_tyAlmText[udiStatus2].sAlmText;

				END_IF

			ELSE
				tyMsgTypeRcv.bBoardForecast := FALSE;
			END_IF

		END_IF

	END_IF

END_ACTION
```

#### Act_Background_Sequence.st - Do Not Change!!!
```iecst
 (** 2021-08-01 **)
ACTION Act_Background_Sequence:

	IF eStatus1 <> Error THEN

		IF p_bOpsRun = FALSE THEN
			p_bRcvIncompl	:= TRUE;
		END_IF

		IF tyMsgTypeRcv.bTransportFinished = TRUE THEN
			IF tyTransportFinished.tyData.eTransferState = HermesTransferStateNotStarted THEN
				p_bRcvNotStart	:= TRUE;
			ELSIF tyTransportFinished.tyData.eTransferState = HermesTransferStateIncomplete THEN
				p_bRcvIncompl	:= TRUE;
			END_IF
		END_IF

		//Sequence
		fbSequenceUS.bRstState		                := bRstState;
		fbSequenceUS.bRdyRcv	                	:= (p_bRdyRcv) AND (eStatus2 <> Error); //Machine in OpsG step USCommTmr (Have USB)
		fbSequenceUS.bBlkUS		                	:= bBlkUS; //Block if different parameter with B.A/B.F(id) Hermes Msg from upstream
		fbSequenceUS.bRdyTransport	                := p_bRdyTransport; //Previously is Always True, now has a 0.1s delay to double check Recipe & Width
		fbSequenceUS.bRcvCompl		                := p_bRcvCompl; //p_bRcvCompl = Pass Inlet Sensor = PCB in Our Machine
		fbSequenceUS.bRcvIncompl	                := p_bRcvIncompl; //Received TransportFinished = Incomplete (Value = 2)
		fbSequenceUS.bRcvNotStart	                := p_bRcvNotStart; //Received TransportFinished = NotStarted (Value = 1)
		fbSequenceUS.bProcessBoardForecastId     	:= bProcessBoardForecastId; //Received BoardForecastId
		fbSequenceUS(bEn := TRUE);
		bNotAvlNotRdy                               := fbSequenceUS.bNotAvlNotRdy;
		bBoardAvailable                             := fbSequenceUS.bBoardAvailable;
		bUSRdy		                               	:= fbSequenceUS.bUSRdy; //bUSRdy:= (eState = HermesStateBoardAvailable) OR (eState = HermesStateAvailableAndReady) OR (eState >= HermesStateTransporting);
		bDSRdy		                               	:= fbSequenceUS.bDSRdy;
		bTransporting                             	:= fbSequenceUS.bTransporting;
		bStopTransport                            	:= fbSequenceUS.bStopTransport;
		bUSGdRdy                                   	:= (tyBoardAvailableRcv.tyAvl.bFailedBoard = FALSE) OR ((tyBoardAvailableRcv.tyAvl.bFailedBoard = TRUE) AND (tyBoardAvailableRcv.tyData.eFailedBoard <> HermesFailedBoard));
		bDSGdRdy                                   	:= (tyMachineReady.tyAvl.bFailedBoard = FALSE) OR ((tyMachineReady.tyAvl.bFailedBoard = TRUE) AND (tyMachineReady.tyData.eFailedBoard <> HermesFailedBoard));

		IF fbSequenceUS.eState >= HermesStateNotAvailableNotReady THEN
			bHandshakeDone	:= TRUE;
		ELSE
			bHandshakeDone	:= FALSE;
		END_IF

		IF EDGEPOS(fbSequenceUS.eState = HermesStateTransporting) THEN
			p_bRcvCompl		:= FALSE;
			p_bRcvIncompl	:= FALSE;
			p_bRcvNotStart	:= FALSE;
		END_IF

		IF fbSequenceUS.eMsgTypeSnd = HermesMsgTypeServiceDescription THEN
			fHermesAddOneMsgSend(ADR(a_eMsgSend) , ADR(udiMsgSendBffr) , HermesMsgTypeServiceDescription);

			tyServiceDescriptionSnd.tyData.sMachineId                                       := p_sMcId;
			tyServiceDescriptionSnd.tyData.iLaneId											:= p_tyParam.iLaneID;
			tyServiceDescriptionSnd.tyData.sInterfaceId										:= p_tyParam.sUpstreamInterfaceId;
			tyServiceDescriptionSnd.tyData.sVersion											:= p_sVersion;
			tyServiceDescriptionSnd.tyData.tySupportedFeatures.bFeatureCheckAliveResponse	:= (p_tyParam.bFeatureCheckAliveResponse) AND (p_tyParam.tRcvAlive <> T#0s) AND (p_tyParam.tSndAlive <> T#0s);
			tyServiceDescriptionSnd.tyData.tySupportedFeatures.bFeatureBoardForecast		:= p_tyParam.bFeatureBoardForecast;
			tyServiceDescriptionSnd.tyData.tySupportedFeatures.bFeatureQueryBoardInfo		:= p_tyParam.bFeatureQueryBoardInfo;
			tyServiceDescriptionSnd.tyData.tySupportedFeatures.bFeatureSendBoardInfo		:= FALSE;

			tyServiceDescriptionSnd.tyAvl.bMachineId										:= TRUE;
			tyServiceDescriptionSnd.tyAvl.bLaneId											:= tyServiceDescriptionSnd.tyData.iLaneId <> 0;
			tyServiceDescriptionSnd.tyAvl.bInterfaceId										:= tyServiceDescriptionSnd.tyData.sInterfaceId <> '';
			tyServiceDescriptionSnd.tyAvl.bVersion											:= TRUE;
			tyServiceDescriptionSnd.tyAvl.bSupportedFeatures								:= p_tyParam.bFeatureCheckAliveResponse OR p_tyParam.bFeatureBoardForecast OR p_tyParam.bFeatureQueryBoardInfo;
			tyServiceDescriptionSnd.tyAvl.tySupportedFeatures.bFeatureCheckAliveResponse	:= (p_tyParam.bFeatureCheckAliveResponse) AND (p_tyParam.tRcvAlive <> T#0s) AND (p_tyParam.tSndAlive <> T#0s);
			tyServiceDescriptionSnd.tyAvl.tySupportedFeatures.bFeatureBoardForecast			:= p_tyParam.bFeatureBoardForecast;
			tyServiceDescriptionSnd.tyAvl.tySupportedFeatures.bFeatureQueryBoardInfo		:= p_tyParam.bFeatureQueryBoardInfo;
			tyServiceDescriptionSnd.tyAvl.tySupportedFeatures.bFeatureSendBoardInfo			:= FALSE;

		ELSIF fbSequenceUS.eMsgTypeSnd = HermesMsgTypeMachineReady THEN
			IF bReplyMcRdyId = FALSE THEN

			    fHermesAddOneMsgSend(ADR(a_eMsgSend) , ADR(udiMsgSendBffr) , HermesMsgTypeMachineReady);

		    	tyMachineReady.tyData.eFailedBoard			:= p_eFailedBoard;
				tyMachineReady.tyAvl.bFailedBoard			:= TRUE;
			    tyMachineReady.tyAvl.bForecastId			:= FALSE;
				tyMachineReady.tyAvl.bBoardId				:= FALSE;
			    tyMachineReady.tyAvl.bProductTypeId			:= FALSE;
			    tyMachineReady.tyAvl.bFlippedBoard			:= FALSE;
			    tyMachineReady.tyAvl.bLength				:= FALSE;
			    tyMachineReady.tyAvl.bWidth					:= FALSE;
			    tyMachineReady.tyAvl.bThickness				:= FALSE;
			    tyMachineReady.tyAvl.bConveyorSpeed			:= FALSE;
			    tyMachineReady.tyAvl.bTopClearanceHeight	:= FALSE;
			    tyMachineReady.tyAvl.bBottomClearanceHeight	:= FALSE;
		    	tyMachineReady.tyAvl.bWeight				:= FALSE;
				tyMachineReady.tyAvl.bWorkOrderId			:= FALSE;
				tyMachineReady.tyAvl.bBatchId    			:= FALSE;

			ELSE
				fHermesAddOneMsgSend(ADR(a_eMsgSend) , ADR(udiMsgSendBffr) , HermesMsgTypeMachineReady);

				tyMachineReady.tyData.eFailedBoard			:= p_eFailedBoard;
				tyMachineReady.tyData.sForecastId	        := tyBoardForecastAcc.tyData.sForecastId;
				tyMachineReady.tyData.sProductTypeId	    := p_sRecipeNm;
				tyMachineReady.tyData.rWidth	            := DINT_TO_REAL(p_diWidthInUM) / 1000;
				tyMachineReady.tyAvl.bFailedBoard			:= TRUE;
				tyMachineReady.tyAvl.bForecastId			:= tyBoardForecastAcc.tyData.sForecastId<>'';
				tyMachineReady.tyAvl.bBoardId				:= FALSE;
				tyMachineReady.tyAvl.bProductTypeId			:= tyBoardForecastAcc.tyData.sProductTypeId<>'';
				tyMachineReady.tyAvl.bFlippedBoard			:= FALSE;
				tyMachineReady.tyAvl.bLength				:= FALSE;
				tyMachineReady.tyAvl.bWidth					:= tyMachineReady.tyData.rWidth<>0;
				tyMachineReady.tyAvl.bThickness				:= FALSE;
				tyMachineReady.tyAvl.bConveyorSpeed			:= FALSE;
				tyMachineReady.tyAvl.bTopClearanceHeight	:= FALSE;
				tyMachineReady.tyAvl.bBottomClearanceHeight	:= FALSE;
				tyMachineReady.tyAvl.bWeight				:= FALSE;
				tyMachineReady.tyAvl.bWorkOrderId			:= FALSE;
				tyMachineReady.tyAvl.bBatchId		    	:= FALSE;

			END_IF

		ELSIF fbSequenceUS.eMsgTypeSnd = HermesMsgTypeRevokeMachineReady THEN
			fHermesAddOneMsgSend(ADR(a_eMsgSend) , ADR(udiMsgSendBffr) , HermesMsgTypeRevokeMachineReady);

		ELSIF fbSequenceUS.eMsgTypeSnd = HermesMsgTypeStartTransport THEN
			fHermesAddOneMsgSend(ADR(a_eMsgSend) , ADR(udiMsgSendBffr) , HermesMsgTypeStartTransport);

			tyStartTransport.tyData.sBoardId		:= tyBoardAvailableRcv.tyData.sBoardId;

			tyStartTransport.tyAvl.bBoardId			:= TRUE;
			tyStartTransport.tyAvl.bConveyorSpeed	:= FALSE;

		ELSIF fbSequenceUS.eMsgTypeSnd = HermesMsgTypeStopTransport THEN
			fHermesAddOneMsgSend(ADR(a_eMsgSend) , ADR(udiMsgSendBffr) , HermesMsgTypeStopTransport);

			IF p_bRcvCompl = TRUE THEN
				tyStopTransport.tyData.eTransferState	:= HermesTransferStateComplete;
			ELSIF p_bRcvIncompl = TRUE THEN
				tyStopTransport.tyData.eTransferState	:= HermesTransferStateIncomplete;
			ELSE
				tyStopTransport.tyData.eTransferState	:= HermesTransferStateNotStarted;
			END_IF
			tyStopTransport.tyData.sBoardId				:= tyStartTransport.tyData.sBoardId;

			tyStopTransport.tyAvl.bTransferState		:= TRUE;
			tyStopTransport.tyAvl.bBoardId				:= TRUE;

		END_IF

	END_IF

END_ACTION
```

#### Act_Background_SequenceTO.st - Do Not Change!!!
```iecst
(** 2021-08-01 **)
ACTION Act_Background_SequenceTO:

	IF (eStatus1 <> Error) AND (eStatus2 <> Error) THEN

		//Time Out
		fbSequenceTO.eState				:= fbSequenceUS.eState;
		fbSequenceTO.tConnTimeOut		:= p_tConnTimeOut;
		fbSequenceTO.tTransportTimeOut	:= DINT_TO_TIME(p_diTransferInTO);
		fbSequenceTO(bEn := TRUE);

		IF fbSequenceTO.udiStatus > 0 AND fbSequenceTO.udiStatus < 65534 THEN

			IF fbSequenceTO.udiStatus = 2912 THEN
				eStatus1	:= Error;
				udiStatus1	:= 10106;	//Service Description Interchange Time Out

				fHermesAddOneMsgSend(ADR(a_eMsgSend) , ADR(udiMsgSendBffr) , HermesMsgTypeNotification);

				tyNotificationSnd.tyAvl.bSeverity			:= TRUE;
				tyNotificationSnd.tyAvl.bNotificationCode	:= TRUE;
				tyNotificationSnd.tyAvl.bDescription		:= TRUE;
				tyNotificationSnd.tyData.eSeverity			:= HermesSeverityFatalError;
				tyNotificationSnd.tyData.iNotificationCode	:= UDINT_TO_INT(udiStatus1);
				tyNotificationSnd.tyData.sDescription		:= a_tyAlmText[udiStatus1].sAlmText;

			ELSIF fbSequenceTO.udiStatus = 2913 THEN
				p_bRcvIncompl	:= TRUE;

				eStatus2	:= Error;
				udiStatus2	:= 10107;	//Transport Time Out

				fHermesAddOneMsgSend(ADR(a_eMsgSend) , ADR(udiMsgSendBffr) , HermesMsgTypeNotification);

				tyNotificationSnd.tyAvl.bSeverity			:= TRUE;
				tyNotificationSnd.tyAvl.bNotificationCode	:= TRUE;
				tyNotificationSnd.tyAvl.bDescription		:= TRUE;
				tyNotificationSnd.tyData.eSeverity			:= HermesSeverityError;
				tyNotificationSnd.tyData.iNotificationCode	:= UDINT_TO_INT(udiStatus2);
				tyNotificationSnd.tyData.sDescription		:= a_tyAlmText[udiStatus2].sAlmText;

			ELSE
				eStatus2	:= Error;
				udiStatus2	:= fbSequenceTO.udiStatus;

				fHermesAddOneMsgSend(ADR(a_eMsgSend) , ADR(udiMsgSendBffr) , HermesMsgTypeNotification);

				tyNotificationSnd.tyAvl.bSeverity			:= TRUE;
				tyNotificationSnd.tyAvl.bNotificationCode	:= TRUE;
				tyNotificationSnd.tyAvl.bDescription		:= TRUE;
				tyNotificationSnd.tyData.eSeverity			:= HermesSeverityFatalError;
				tyNotificationSnd.tyData.iNotificationCode	:= UDINT_TO_INT(udiStatus2);
				tyNotificationSnd.tyData.sDescription		:= a_tyAlmText[udiStatus2].sAlmText;

			END_IF

		END_IF

	END_IF

END_ACTION
```

#### Act_Background_BoardAvailableChk.st - Do Not Change!!!
```iecst
(** 2021-08-01 **)
ACTION Act_Background_BoardAvailableChk:

	IF eStatus2 <> Error THEN
		IF p_bNewIncomingBoard = FALSE AND p_bSiemensMcModeChgPrep = FALSE AND (bTransporting = FALSE) AND(p_bOpsRun = TRUE) THEN
			bBaReceivedInRdyState	:= p_bAccDataRdy AND (bTransporting = FALSE) AND(p_bOpsRun = TRUE);//AutoRcp
			bAccDataReq		:= FALSE;
			bBABlkUS		:= FALSE;
			bOverWriteSlt	:= FALSE;
			bOverWriteWidth	:= FALSE;

			IF p_tyParam.bCmpTypeId = TRUE  THEN	//"Compare Type ID" Ticked

				IF tyBoardAvailableRcv.tyAvl.bProductTypeId = TRUE THEN	//Check if there is Product Type Id in B.A msg

					IF tyBoardAvailableRcv.tyData.sProductTypeId <> p_sRecipeNm THEN	//Product Type Id Different

						bAccDataReq	    := TRUE;	//Require To Load New Recipe
						bBABlkUS		:= TRUE;

						sReqRecipeNm	:= tyBoardAvailableRcv.tyData.sProductTypeId;
						diReqWidthInUM	:= REAL_TO_DINT(tyBoardAvailableRcv.tyData.rWidth * 1000);

					ELSE	//Product Type Id Same (After accepted or Originally same)

						IF p_tyParam.bCmpParam = TRUE THEN	//"Compare Param" Ticked
							IF tyBoardAvailableRcv.tyAvl.bThickness AND tyBoardAvailableRcv.tyAvl.bTopClearanceHeight AND tyBoardAvailableRcv.tyAvl.bBottomClearanceHeight AND p_bBASltEn THEN	//Camparing Slot Parameters if p_bBASltEn = TRUE
								udiStatus2	:= fHermesCmpSlt(tyBoardAvailableRcv.tyData.eFlippedBoard , tyBoardAvailableRcv.tyData.rThickness , tyBoardAvailableRcv.tyData.rTopClearanceHeight , tyBoardAvailableRcv.tyData.rBottomClearanceHeight , p_diMinSltValue , p_diMaxSltValue , p_diPitch , p_diSltToSltInUM , p_diTtlSlt);

								IF udiStatus2 <> 0 THEN

									bBABlkUS	:= TRUE;

									eStatus2	:= Error;

									IF udiStatus2 = 2914 THEN
										udiStatus2	:= 10108;	//Input First Slot Is Invalid
									ELSIF udiStatus2 = 2915 THEN
										udiStatus2	:= 10109;	//Input Last Slot Is Invalid
									ELSIF udiStatus2 = 2916 THEN
										udiStatus2	:= 10110;	//Input Pitch Is Invalid
									ELSIF udiStatus2 = 2917 THEN
										udiStatus2	:= 10111;	//Input Slot To Slot Distance Is Invalid
									ELSIF udiStatus2 = 2918 THEN
										udiStatus2	:= 10112;	//Input Total Slot Is Invalid
									ELSIF udiStatus2 = 2919 THEN
										udiStatus2	:= 10113;	//Input Thickness Is Invalid
									ELSIF udiStatus2 = 2920 THEN
										udiStatus2	:= 10114;	//Input Top Clearance Height Is Invalid
									ELSIF udiStatus2 = 2921 THEN
										udiStatus2	:= 10115;	//Input Bottom Clearance Height Is Invalid
									ELSIF udiStatus2 = 2922 THEN
										udiStatus2	:= 10116;	//Recipe First Slot Value & Board Available Data Not Match With Same Product Type Id
									ELSIF udiStatus2 = 2923 THEN
										udiStatus2	:= 10117;	//Recipe Last Slot Value & Board Available Data Not Match With Same Product Type Id
									ELSIF udiStatus2 = 2924 THEN
										udiStatus2	:= 10118;	//Recipe Pitch Value & Board Available Data Not Match With Same Product Type Id
									END_IF

									fHermesAddOneMsgSend(ADR(a_eMsgSend) , ADR(udiMsgSendBffr) , HermesMsgTypeNotification);

									tyNotificationSnd.tyAvl.bSeverity			:= TRUE;
									tyNotificationSnd.tyAvl.bNotificationCode	:= TRUE;
									tyNotificationSnd.tyAvl.bDescription		:= TRUE;
									tyNotificationSnd.tyData.eSeverity			:= HermesSeverityError;
									tyNotificationSnd.tyData.iNotificationCode	:= UDINT_TO_INT(udiStatus2);
									tyNotificationSnd.tyData.sDescription		:= a_tyAlmText[udiStatus2].sAlmText;

								END_IF
							END_IF

							IF tyBoardAvailableRcv.tyAvl.bWidth AND p_bBAWidthEn THEN	//Comparing Width Parameter if p_bBAWidthEn = TRUE
								IF REAL_TO_DINT(tyBoardAvailableRcv.tyData.rWidth * 1000) <> p_diWidthInUM THEN

									bBABlkUS	:= TRUE;

									eStatus2	:= Error;
									udiStatus2	:= 10119;	//Width Different With Same Product Type Id

									fHermesAddOneMsgSend(ADR(a_eMsgSend) , ADR(udiMsgSendBffr) , HermesMsgTypeNotification);

									tyNotificationSnd.tyAvl.bSeverity			:= TRUE;
									tyNotificationSnd.tyAvl.bNotificationCode	:= TRUE;
									tyNotificationSnd.tyAvl.bDescription		:= TRUE;
									tyNotificationSnd.tyData.eSeverity			:= HermesSeverityError;
									tyNotificationSnd.tyData.iNotificationCode	:= UDINT_TO_INT(udiStatus2);
									tyNotificationSnd.tyData.sDescription		:= a_tyAlmText[udiStatus2].sAlmText;

								END_IF
							END_IF

						END_IF

					END_IF

				ELSE

					eStatus2	:= Error;
					udiStatus2	:= 10158;	//Product Type Id Not Receive From Upstream

					fHermesAddOneMsgSend(ADR(a_eMsgSend) , ADR(udiMsgSendBffr) , HermesMsgTypeNotification);

					tyNotificationSnd.tyAvl.bSeverity			:= TRUE;
					tyNotificationSnd.tyAvl.bNotificationCode	:= TRUE;
					tyNotificationSnd.tyAvl.bDescription		:= TRUE;
					tyNotificationSnd.tyData.eSeverity			:= HermesSeverityError;
					tyNotificationSnd.tyData.iNotificationCode	:= UDINT_TO_INT(udiStatus2);
					tyNotificationSnd.tyData.sDescription		:= a_tyAlmText[udiStatus2].sAlmText;

				END_IF

			ELSE	//"Compare Type ID" Not Ticked
				                                    //Add
				IF p_tyParam.bOverwrite AND p_bNewIncomingBoard = FALSE  THEN	//"Overwrite" Ticked

					IF tyBoardAvailableRcv.tyAvl.bThickness AND tyBoardAvailableRcv.tyAvl.bTopClearanceHeight AND tyBoardAvailableRcv.tyAvl.bBottomClearanceHeight AND p_bBASltEn THEN	//Camparing Slot Parameters

						udiStatus2	:= fHermesCmpSlt(tyBoardAvailableRcv.tyData.eFlippedBoard , tyBoardAvailableRcv.tyData.rThickness , tyBoardAvailableRcv.tyData.rTopClearanceHeight , tyBoardAvailableRcv.tyData.rBottomClearanceHeight , p_diMinSltValue , p_diMaxSltValue , p_diPitch , p_diSltToSltInUM , p_diTtlSlt);

						IF udiStatus2 <> 0 THEN

							bAccDataReq		:= TRUE;
							bBABlkUS			:= TRUE;
							bOverWriteSlt	:= TRUE;

							fbGetSlt.eFlippedBrd				:= tyBoardAvailableRcv.tyData.eFlippedBoard;
							fbGetSlt.rThicknessInMM				:= tyBoardAvailableRcv.tyData.rThickness;
							fbGetSlt.rTopClearanceHeightInMM	:= tyBoardAvailableRcv.tyData.rTopClearanceHeight;
							fbGetSlt.rBtmClearanceHeightInMM	:= tyBoardAvailableRcv.tyData.rBottomClearanceHeight;
							fbGetSlt.diSltToSltInUM				:= p_diSltToSltInUM;
							fbGetSlt.diTtlSlt					:= p_diTtlSlt;
							fbGetSlt;

							diReqMinSltValue	:= fbGetSlt.diMinSltValue;
							diReqMaxSltValue	:= fbGetSlt.diMaxSltValue;
							diReqPitch			:= fbGetSlt.diPitch;

						END_IF

					END_IF

					IF tyBoardAvailableRcv.tyAvl.bWidth  AND p_bBAWidthEn AND p_usiLinkProdRcpCurrRcpMcMod = 0 THEN	//Comparing Width Parameter
						IF REAL_TO_DINT(tyBoardAvailableRcv.tyData.rWidth * 1000) <> p_diWidthInUM THEN

							bAccDataReq		:= TRUE;
							bBABlkUS		:= TRUE;
							bOverWriteWidth	:= TRUE;

							diReqWidthInUM	:= REAL_TO_DINT(tyBoardAvailableRcv.tyData.rWidth * 1000);

						END_IF
					END_IF

				ELSE	//"Compare Type ID" Not Ticked and "Overwrite" Not Ticked, Error if not same

					IF tyBoardAvailableRcv.tyAvl.bThickness AND tyBoardAvailableRcv.tyAvl.bTopClearanceHeight AND tyBoardAvailableRcv.tyAvl.bBottomClearanceHeight AND p_bBASltEn AND p_bRdyRcv THEN	//Camparing Slot Parameters
						udiStatus2	:= fHermesCmpSlt(tyBoardAvailableRcv.tyData.eFlippedBoard , tyBoardAvailableRcv.tyData.rThickness , tyBoardAvailableRcv.tyData.rTopClearanceHeight , tyBoardAvailableRcv.tyData.rBottomClearanceHeight , p_diMinSltValue , p_diMaxSltValue , p_diPitch , p_diSltToSltInUM , p_diTtlSlt);

						IF udiStatus2 <> 0 THEN

							bBABlkUS		:= TRUE;

							eStatus2	:= Error;

							IF udiStatus2 = 2914 THEN
								udiStatus2	:= 10120;	//Input First Slot Is Invalid
							ELSIF udiStatus2 = 2915 THEN
								udiStatus2	:= 10121;	//Input Last Slot Is Invalid
							ELSIF udiStatus2 = 2916 THEN
								udiStatus2	:= 10122;	//Input Pitch Is Invalid
							ELSIF udiStatus2 = 2917 THEN
								udiStatus2	:= 10123;	//Input Slot To Slot Distance Is Invalid
							ELSIF udiStatus2 = 2918 THEN
								udiStatus2	:= 10124;	//Input Total Slot Is Invalid
							ELSIF udiStatus2 = 2919 THEN
								udiStatus2	:= 10125;	//Input Thickness Is Invalid
							ELSIF udiStatus2 = 2920 THEN
								udiStatus2	:= 10126;	//Input Top Clearance Height Is Invalid
							ELSIF udiStatus2 = 2921 THEN
								udiStatus2	:= 10127;	//Input Bottom Clearance Height Is Invalid
							ELSIF udiStatus2 = 2922 THEN
								udiStatus2	:= 10128;	//Recipe First Slot Value & Board Available Data Not Match With Same Product Type Id
							ELSIF udiStatus2 = 2923 THEN
								udiStatus2	:= 10129;	//Recipe Last Slot Value & Board Available Data Not Match With Same Product Type Id
							ELSIF udiStatus2 = 2924 THEN
								udiStatus2	:= 10130;	//Recipe Pitch Value & Board Available Data Not Match With Same Product Type Id
							END_IF

							fHermesAddOneMsgSend(ADR(a_eMsgSend) , ADR(udiMsgSendBffr) , HermesMsgTypeNotification);

							tyNotificationSnd.tyAvl.bSeverity			:= TRUE;
							tyNotificationSnd.tyAvl.bNotificationCode	:= TRUE;
							tyNotificationSnd.tyAvl.bDescription		:= TRUE;
							tyNotificationSnd.tyData.eSeverity			:= HermesSeverityError;
							tyNotificationSnd.tyData.iNotificationCode	:= UDINT_TO_INT(udiStatus2);
							tyNotificationSnd.tyData.sDescription		:= a_tyAlmText[udiStatus2].sAlmText;

						END_IF
					END_IF

					IF tyBoardAvailableRcv.tyAvl.bWidth AND p_bBAWidthEn AND p_bRdyRcv THEN	//Comparing Width Parameter
						IF REAL_TO_DINT(tyBoardAvailableRcv.tyData.rWidth * 1000) <> p_diWidthInUM THEN

							bBABlkUS		:= TRUE;

							eStatus2	:= Error;
							udiStatus2	:= 10131;	//Width Different With Same Product Type Id

							fHermesAddOneMsgSend(ADR(a_eMsgSend) , ADR(udiMsgSendBffr) , HermesMsgTypeNotification);

							tyNotificationSnd.tyAvl.bSeverity			:= TRUE;
							tyNotificationSnd.tyAvl.bNotificationCode	:= TRUE;
							tyNotificationSnd.tyAvl.bDescription		:= TRUE;
							tyNotificationSnd.tyData.eSeverity			:= HermesSeverityError;
							tyNotificationSnd.tyData.iNotificationCode	:= UDINT_TO_INT(udiStatus2);
							tyNotificationSnd.tyData.sDescription		:= a_tyAlmText[udiStatus2].sAlmText;

						END_IF
					END_IF

				END_IF

			END_IF

		ELSIF (p_bAccDataRdy = FALSE) OR bTransporting = TRUE THEN

			bAccDataReq		:= FALSE;
			bBABlkUS		:= FALSE;
			bOverWriteSlt	:= FALSE;
			bOverWriteWidth	:= FALSE;

		END_IF

	ELSE

		bAccDataReq		:= FALSE;
		bBABlkUS		:= TRUE;
		bOverWriteSlt	:= FALSE;
		bOverWriteWidth	:= FALSE;

	END_IF

END_ACTION
```

#### Act_Background_BoardForecastIdChk.st - Do Not Change!!!
```iecst
(** 2021-08-01 **)
ACTION Act_Background_BoardForecastIdChk:

	IF eStatus2 <> Error  THEN

		IF bProcessBoardForecastId AND bNotAvlNotRdy AND (bTransporting = FALSE) AND (p_bOpsRun = TRUE) AND p_bSiemensMcModeChgPrep = FALSE THEN
			bBfReceivedInRdyState := 	bProcessBoardForecastId AND bNotAvlNotRdy AND (bTransporting = FALSE) AND (p_bOpsRun = TRUE)  ;	 //AutoRcp
			bBFAccDataReq		:= FALSE;
			bBFBlkUS			:= FALSE;
			bBFOverWriteSlt  	:= FALSE;
			bBFOverWriteWidth	:= FALSE;
			                                      //Add
			IF p_tyParam.bCmpTypeId = TRUE AND p_bNewIncomingBoard = FALSE  THEN	//"Compare Type ID" Ticked

				IF tyBoardForecastAcc.tyAvl.bProductTypeId = TRUE THEN	//Check if there is Product Type Id in B.F msg

					IF tyBoardForecastAcc.tyData.sProductTypeId <> p_sRecipeNm THEN	//Product Type Id Different

						bBFAccDataReq	:= TRUE;	//Require To Load New Recipe
						bBFBlkUS		:= TRUE;

						sReqRecipeNm	:= tyBoardForecastAcc.tyData.sProductTypeId;
						diReqWidthInUM	:= REAL_TO_DINT(tyBoardForecastAcc.tyData.rWidth * 1000);

					ELSE	//Product Type Id Same (After accepted or Originally same)

						IF p_tyParam.bCmpParam = TRUE THEN	//"Compare Param" Ticked
							IF tyBoardForecastAcc.tyAvl.bThickness AND tyBoardForecastAcc.tyAvl.bTopClearanceHeight AND tyBoardForecastAcc.tyAvl.bBottomClearanceHeight AND p_bBFSltEn THEN	//Camparing Slot Parameters if p_bBFSltEn = TRUE
								udiStatus2	:= fHermesCmpSlt(tyBoardForecastAcc.tyData.eFlippedBoard , tyBoardForecastAcc.tyData.rThickness , tyBoardForecastAcc.tyData.rTopClearanceHeight , tyBoardForecastAcc.tyData.rBottomClearanceHeight , p_diMinSltValue , p_diMaxSltValue , p_diPitch , p_diSltToSltInUM , p_diTtlSlt);

								IF udiStatus2 <> 0 THEN

									bBFBlkUS		:= TRUE;
									bProcessBoardForecastId := FALSE;//add
									eStatus2	:= Error;

									IF udiStatus2 = 2914 THEN
										udiStatus2	:= 10108;	//Input First Slot Is Invalid
									ELSIF udiStatus2 = 2915 THEN
										udiStatus2	:= 10109;	//Input Last Slot Is Invalid
									ELSIF udiStatus2 = 2916 THEN
										udiStatus2	:= 10110;	//Input Pitch Is Invalid
									ELSIF udiStatus2 = 2917 THEN
										udiStatus2	:= 10111;	//Input Slot To Slot Distance Is Invalid
									ELSIF udiStatus2 = 2918 THEN
										udiStatus2	:= 10112;	//Input Total Slot Is Invalid
									ELSIF udiStatus2 = 2919 THEN
										udiStatus2	:= 10113;	//Input Thickness Is Invalid
									ELSIF udiStatus2 = 2920 THEN
										udiStatus2	:= 10114;	//Input Top Clearance Height Is Invalid
									ELSIF udiStatus2 = 2921 THEN
										udiStatus2	:= 10115;	//Input Bottom Clearance Height Is Invalid
									ELSIF udiStatus2 = 2922 THEN
										udiStatus2	:= 10116;	//Recipe First Slot Value & Board Available Data Not Match With Same Product Type Id
									ELSIF udiStatus2 = 2923 THEN
										udiStatus2	:= 10117;	//Recipe Last Slot Value & Board Available Data Not Match With Same Product Type Id
									ELSIF udiStatus2 = 2924 THEN
										udiStatus2	:= 10118;	//Recipe Pitch Value & Board Available Data Not Match With Same Product Type Id
									END_IF

									fHermesAddOneMsgSend(ADR(a_eMsgSend) , ADR(udiMsgSendBffr) , HermesMsgTypeNotification);

									tyNotificationSnd.tyAvl.bSeverity			:= TRUE;
									tyNotificationSnd.tyAvl.bNotificationCode	:= TRUE;
									tyNotificationSnd.tyAvl.bDescription		:= TRUE;
									tyNotificationSnd.tyData.eSeverity			:= HermesSeverityError;
									tyNotificationSnd.tyData.iNotificationCode	:= 6; //BoardForecast Error
									tyNotificationSnd.tyData.sDescription		:= a_tyAlmText[udiStatus2].sAlmText;

								END_IF
							END_IF

							IF tyBoardForecastAcc.tyAvl.bWidth AND p_bBFWidthEn THEN	//Comparing Width Parameter if p_bBFWidthEn = TRUE
								IF REAL_TO_DINT(tyBoardForecastAcc.tyData.rWidth * 1000) <> p_diWidthInUM THEN

									bBFBlkUS	:= TRUE;
									bProcessBoardForecastId := FALSE;//add
									eStatus2	:= Error;
									udiStatus2	:= 10119;	//Width Different With Same Product Type Id

									fHermesAddOneMsgSend(ADR(a_eMsgSend) , ADR(udiMsgSendBffr) , HermesMsgTypeNotification);

									tyNotificationSnd.tyAvl.bSeverity			:= TRUE;
									tyNotificationSnd.tyAvl.bNotificationCode	:= TRUE;
									tyNotificationSnd.tyAvl.bDescription		:= TRUE;
									tyNotificationSnd.tyData.eSeverity			:= HermesSeverityError;
									tyNotificationSnd.tyData.iNotificationCode	:= 6; //BoardForecast Error
									tyNotificationSnd.tyData.sDescription		:= a_tyAlmText[udiStatus2].sAlmText;
								ELSE
									bReplyMcRdyId           := TRUE; //add
									bProcessBoardForecastId := FALSE; //add
								END_IF
							END_IF

						END_IF

					END_IF

				ELSE

					eStatus2	:= Error;
					udiStatus2	:= 10158;	//Product Type Id Not Receive From Upstream
					bProcessBoardForecastId := FALSE;//add

					fHermesAddOneMsgSend(ADR(a_eMsgSend) , ADR(udiMsgSendBffr) , HermesMsgTypeNotification);

					tyNotificationSnd.tyAvl.bSeverity			:= TRUE;
					tyNotificationSnd.tyAvl.bNotificationCode	:= TRUE;
					tyNotificationSnd.tyAvl.bDescription		:= TRUE;
					tyNotificationSnd.tyData.eSeverity			:= HermesSeverityError;
					tyNotificationSnd.tyData.iNotificationCode	:= 6; //BoardForecast Error
					tyNotificationSnd.tyData.sDescription		:= a_tyAlmText[udiStatus2].sAlmText;

				END_IF

			ELSE	//"Compare Type ID" Not Ticked

				IF p_tyParam.bOverwrite AND p_bNewIncomingBoard = FALSE   THEN	//"Overwrite" Ticked

					IF tyBoardForecastAcc.tyAvl.bThickness AND tyBoardForecastAcc.tyAvl.bTopClearanceHeight AND tyBoardForecastAcc.tyAvl.bBottomClearanceHeight AND p_bBFSltEn THEN	//Camparing Slot Parameters

						udiStatus2	:= fHermesCmpSlt(tyBoardForecastAcc.tyData.eFlippedBoard , tyBoardForecastAcc.tyData.rThickness , tyBoardForecastAcc.tyData.rTopClearanceHeight , tyBoardForecastAcc.tyData.rBottomClearanceHeight , p_diMinSltValue , p_diMaxSltValue , p_diPitch , p_diSltToSltInUM , p_diTtlSlt);

						IF udiStatus2 <> 0 THEN

							bBFAccDataReq		:= TRUE;
							bBFBlkUS			:= TRUE;
							bBFOverWriteSlt	    := TRUE;

							fbGetSlt.eFlippedBrd				:= tyBoardForecastAcc.tyData.eFlippedBoard;
							fbGetSlt.rThicknessInMM				:= tyBoardForecastAcc.tyData.rThickness;
							fbGetSlt.rTopClearanceHeightInMM	:= tyBoardForecastAcc.tyData.rTopClearanceHeight;
							fbGetSlt.rBtmClearanceHeightInMM	:= tyBoardForecastAcc.tyData.rBottomClearanceHeight;
							fbGetSlt.diSltToSltInUM				:= p_diSltToSltInUM;
							fbGetSlt.diTtlSlt					:= p_diTtlSlt;
							fbGetSlt;

							diReqMinSltValue	:= fbGetSlt.diMinSltValue;
							diReqMaxSltValue	:= fbGetSlt.diMaxSltValue;
							diReqPitch			:= fbGetSlt.diPitch;

						END_IF

					END_IF

					IF tyBoardForecastAcc.tyAvl.bWidth AND p_bBFWidthEn THEN	//Comparing Width Parameter
						IF REAL_TO_DINT(tyBoardForecastAcc.tyData.rWidth * 1000) <> p_diWidthInUM THEN

							bBFAccDataReq		:= TRUE;
							bBFBlkUS			:= TRUE;
							bBFOverWriteWidth	:= TRUE;

							diReqWidthInUM	:= REAL_TO_DINT(tyBoardForecastAcc.tyData.rWidth * 1000);
						ELSE
							bReplyMcRdyId           := TRUE; //add
							bProcessBoardForecastId := FALSE; //add
						END_IF
					END_IF

				ELSE	//"Compare Type ID" Not Ticked and "Overwrite" Not Ticked, Error if not same

					IF tyBoardForecastAcc.tyAvl.bThickness AND tyBoardForecastAcc.tyAvl.bTopClearanceHeight AND tyBoardForecastAcc.tyAvl.bBottomClearanceHeight AND p_bBFSltEn AND p_bRdyRcv THEN	//Camparing Slot Parameters
						udiStatus2	:= fHermesCmpSlt(tyBoardForecastAcc.tyData.eFlippedBoard , tyBoardForecastAcc.tyData.rThickness , tyBoardForecastAcc.tyData.rTopClearanceHeight , tyBoardForecastAcc.tyData.rBottomClearanceHeight , p_diMinSltValue , p_diMaxSltValue , p_diPitch , p_diSltToSltInUM , p_diTtlSlt);

						IF udiStatus2 <> 0 THEN

							bBFBlkUS		:= TRUE;
							bProcessBoardForecastId := FALSE;//add
							eStatus2	:= Error;

							IF udiStatus2 = 2914 THEN
								udiStatus2	:= 10120;	//Input First Slot Is Invalid
							ELSIF udiStatus2 = 2915 THEN
								udiStatus2	:= 10121;	//Input Last Slot Is Invalid
							ELSIF udiStatus2 = 2916 THEN
								udiStatus2	:= 10122;	//Input Pitch Is Invalid
							ELSIF udiStatus2 = 2917 THEN
								udiStatus2	:= 10123;	//Input Slot To Slot Distance Is Invalid
							ELSIF udiStatus2 = 2918 THEN
								udiStatus2	:= 10124;	//Input Total Slot Is Invalid
							ELSIF udiStatus2 = 2919 THEN
								udiStatus2	:= 10125;	//Input Thickness Is Invalid
							ELSIF udiStatus2 = 2920 THEN
								udiStatus2	:= 10126;	//Input Top Clearance Height Is Invalid
							ELSIF udiStatus2 = 2921 THEN
								udiStatus2	:= 10127;	//Input Bottom Clearance Height Is Invalid
							ELSIF udiStatus2 = 2922 THEN
								udiStatus2	:= 10128;	//Recipe First Slot Value & Board Available Data Not Match With Same Product Type Id
							ELSIF udiStatus2 = 2923 THEN
								udiStatus2	:= 10129;	//Recipe Last Slot Value & Board Available Data Not Match With Same Product Type Id
							ELSIF udiStatus2 = 2924 THEN
								udiStatus2	:= 10130;	//Recipe Pitch Value & Board Available Data Not Match With Same Product Type Id
							END_IF

							fHermesAddOneMsgSend(ADR(a_eMsgSend) , ADR(udiMsgSendBffr) , HermesMsgTypeNotification);

							tyNotificationSnd.tyAvl.bSeverity			:= TRUE;
							tyNotificationSnd.tyAvl.bNotificationCode	:= TRUE;
							tyNotificationSnd.tyAvl.bDescription		:= TRUE;
							tyNotificationSnd.tyData.eSeverity			:= HermesSeverityError;
							tyNotificationSnd.tyData.iNotificationCode	:= 6; //BoardForecast Error
							tyNotificationSnd.tyData.sDescription		:= a_tyAlmText[udiStatus2].sAlmText;

						END_IF
					END_IF

					IF tyBoardForecastAcc.tyAvl.bWidth AND p_bBFWidthEn AND p_bRdyRcv THEN	//Comparing Width Parameter
						IF REAL_TO_DINT(tyBoardForecastAcc.tyData.rWidth * 1000) <> p_diWidthInUM THEN

							bBFBlkUS		:= TRUE;
							bProcessBoardForecastId := FALSE;//add
							eStatus2	:= Error;
							udiStatus2	:= 10131;	//Width Different With Same Product Type Id

							fHermesAddOneMsgSend(ADR(a_eMsgSend) , ADR(udiMsgSendBffr) , HermesMsgTypeNotification);

							tyNotificationSnd.tyAvl.bSeverity			:= TRUE;
							tyNotificationSnd.tyAvl.bNotificationCode	:= TRUE;
							tyNotificationSnd.tyAvl.bDescription		:= TRUE;
							tyNotificationSnd.tyData.eSeverity			:= HermesSeverityError;
							tyNotificationSnd.tyData.iNotificationCode	:= 6; //BoardForecast Error
							tyNotificationSnd.tyData.sDescription		:= a_tyAlmText[udiStatus2].sAlmText;
						ELSE
							bReplyMcRdyId           := TRUE; //add
							bProcessBoardForecastId := FALSE; //add
						END_IF
					END_IF

				END_IF

			END_IF

		ELSIF bProcessBoardForecastId = FALSE OR bNotAvlNotRdy =FALSE OR bTransporting = TRUE THEN

			bBFAccDataReq		:= FALSE;
			bBFBlkUS			:= FALSE;
			bBFOverWriteSlt	    := FALSE;
			bBFOverWriteWidth	:= FALSE;

		END_IF

	ELSE

		bBFAccDataReq		:= FALSE;
		bBFBlkUS			:= TRUE;
		bBFOverWriteSlt	    := FALSE;
		bBFOverWriteWidth	:= FALSE;

	END_IF

END_ACTION
```

#### Act_Background_ChgConfig.st - Do Not Change!!!
```iecst
(** 2021-08-01 **)
ACTION Act_Background_ChgConfig:

	IF eStatus2 <> Error THEN

		IF (tyParamOld.iLaneID <> p_tyParam.iLaneID) OR (tyParamOld.sHostAddress <> p_tyParam.sHostAddress) OR (tyParamOld.uiHostPort <> p_tyParam.uiHostPort)
			OR (tyParamOld.bFeatureBoardForecast <> p_tyParam.bFeatureBoardForecast) OR (tyParamOld.bFeatureCheckAliveResponse <> p_tyParam.bFeatureCheckAliveResponse) OR (tyParamOld.bFeatureQueryBoardInfo <> p_tyParam.bFeatureQueryBoardInfo) THEN

			fHermesAddOneMsgSend(ADR(a_eMsgSend) , ADR(udiMsgSendBffr) , HermesMsgTypeNotification);

			tyNotificationSnd.tyAvl.bSeverity			:= TRUE;
			tyNotificationSnd.tyAvl.bNotificationCode	:= TRUE;
			tyNotificationSnd.tyAvl.bDescription		:= TRUE;
			tyNotificationSnd.tyData.eSeverity			:= HermesSeverityFatalError;
			tyNotificationSnd.tyData.iNotificationCode	:= 3;
			tyNotificationSnd.tyData.sDescription		:= 'Configuration Changed';

			bRstConnection	:= TRUE;

		END_IF

	END_IF

END_ACTION
```

#### Act_Background_QueryBoardInfo.st - Do Not Change!!!
```iecst
(** 2021-08-01 **)
ACTION Act_Background_QueryBoardInfo:

	IF eStatus2 <> Error THEN

		IF EDGEPOS(p_bQueryBoardInfo) THEN

			fHermesAddOneMsgSend(ADR(a_eMsgSend) , ADR(udiMsgSendBffr) , HermesMsgTypeQueryBoardInfo);

			tyQueryBoardInfo.tyData.sTopBarcode						            := p_sTopBarcode;
			tyQueryBoardInfo.tyData.sBottomBarcode							    := p_sBottomBarcode;

			tyQueryBoardInfo.tyAvl.bTopBarcode									:= tyQueryBoardInfo.tyData.sTopBarcode <> '';
			tyQueryBoardInfo.tyAvl.bBottomBarcode							    := tyQueryBoardInfo.tyData.sBottomBarcode <>'';

		END_IF

		IF tyMsgTypeRcv.bSendBoardInfo THEN

			IF p_bQueryBoardInfo AND (udiStatus2 = 0) THEN //After CmpParamRcv
				IF tySendBoardInfoRcv.tyAvl.bBoardId AND tySendBoardInfoRcv.tyAvl.bBoardIdCreatedBy THEN; // AND p_bManualInsertZoneHvBrd = FALSE AND p_bManualInsertEndSen = FALSE THEN //Wait Empty

					bRcvBoardInfoOk              := TRUE;
					tySendBoardInfoAcc          := tySendBoardInfoRcv;
					tyMsgTypeRcv.bSendBoardInfo := FALSE;

				ELSIF ((tySendBoardInfoRcv.tyAvl.bBoardId = FALSE) OR (tySendBoardInfoRcv.tyAvl.bBoardIdCreatedBy = FALSE)) THEN //no BoardId or BoardIdCreatedBy
					bRcvBoardInfoIncompl := TRUE;
					bManuallInsertLastZone         := FALSE;
					tyMsgTypeRcv.bSendBoardInfo := FALSE;
				END_IF

			ELSIF p_bQueryBoardInfo = FALSE THEN
				tyMsgTypeRcv.bSendBoardInfo     := FALSE;
			END_IF

		END_IF

		IF 	bRcvBoardInfoOk = TRUE THEN
			bManuallInsertLastZone        := TRUE; //Board data received from upstream, block Upstream to allow manual insert

			tyInfoData1.sProgNm		:= p_sProgNm;
			tyInfoData1.udiCode		:= 10000;
			tyInfoData1.eSeverity	:= AlmSeverityInfo;
			tyInfoData1.sAlmMsg		:= p_sInfoMsg1;

			IF p_bTransportFinished   THEN

				bRcvBoardInfoOk := FALSE;
				bManuallInsertLastZone        := FALSE;
			END_IF

		ELSIF bRcvBoardInfoIncompl = TRUE THEN //receive dummy, no need block upstream

			tyInfoData2.sProgNm		:= p_sProgNm;
			tyInfoData2.udiCode		:= 10000;
			tyInfoData2.eSeverity	:= AlmSeverityInfo;
			tyInfoData2.sAlmMsg		:= p_sInfoMsg2;

		END_IF

		IF p_bQueryBoardInfo = FALSE THEN

			//Clear Info Message 1
			tyInfoData1.sProgNm		:= '';
			tyInfoData1.udiCode		:= 0;
			tyInfoData1.eSeverity	:= AlmSeverityNA;
			tyInfoData1.sAlmMsg		:= '';
			bRcvBoardInfoOk := FALSE;
			bManuallInsertLastZone        := FALSE;

			//Clear Info Message 2
			tyInfoData2.sProgNm		:= '';
			tyInfoData2.udiCode		:= 0;
			tyInfoData2.eSeverity	:= AlmSeverityNA;
			tyInfoData2.sAlmMsg		:= '';
			bRcvBoardInfoIncompl := FALSE;

		END_IF

	END_IF

END_ACTION
```

#### Act_Background_TCPSend.st - Do Not Change!!!
```iecst
(** 2021-08-01 **)
ACTION Act_Background_TCPSend:

	//Message Send (Generate XML Message)
	IF a_eMsgSend[0] <> HermesMsgTypeNA THEN

		IF a_eMsgSend[0] = HermesMsgTypeCheckAlive THEN
			fHermesFormCheckAlive(ADR(a_tyXMLTableDataSnd) , p_tyDTStructure , tyCheckAliveSnd);
			fTableConvertToXML(ADR(sSnd) , ADR(udiSndMsgLen) , SIZEOF(sSnd) , ADR(a_tyXMLTableDataSnd) , ADR(a_tyXMLTableDataSnd[0].sTitle) , ADR(a_tyXMLTableDataSnd[0].sValue) , ADR(a_tyXMLTableDataSnd[0].uiSize) , SIZEOF(a_tyXMLTableDataSnd[0]) , 12);

		ELSIF a_eMsgSend[0] = HermesMsgTypeCheckAlivePing THEN
			fHermesFormCheckAlive(ADR(a_tyXMLTableDataSnd) , p_tyDTStructure , tyCheckAlivePingSnd);
			fTableConvertToXML(ADR(sSnd) , ADR(udiSndMsgLen) , SIZEOF(sSnd) , ADR(a_tyXMLTableDataSnd) , ADR(a_tyXMLTableDataSnd[0].sTitle) , ADR(a_tyXMLTableDataSnd[0].sValue) , ADR(a_tyXMLTableDataSnd[0].uiSize) , SIZEOF(a_tyXMLTableDataSnd[0]) , 12);

		ELSIF a_eMsgSend[0] = HermesMsgTypeCheckAlivePong THEN
			fHermesFormCheckAlive(ADR(a_tyXMLTableDataSnd) , p_tyDTStructure , tyCheckAlivePongSnd);
			fTableConvertToXML(ADR(sSnd) , ADR(udiSndMsgLen) , SIZEOF(sSnd) , ADR(a_tyXMLTableDataSnd) , ADR(a_tyXMLTableDataSnd[0].sTitle) , ADR(a_tyXMLTableDataSnd[0].sValue) , ADR(a_tyXMLTableDataSnd[0].uiSize) , SIZEOF(a_tyXMLTableDataSnd[0]) , 12);

		ELSIF a_eMsgSend[0] = HermesMsgTypeServiceDescription THEN
			fHermesFormServiceDescription(ADR(a_tyXMLTableDataSnd) , p_tyDTStructure , tyServiceDescriptionSnd);
			fTableConvertToXML(ADR(sSnd) , ADR(udiSndMsgLen) , SIZEOF(sSnd) , ADR(a_tyXMLTableDataSnd) , ADR(a_tyXMLTableDataSnd[0].sTitle) , ADR(a_tyXMLTableDataSnd[0].sValue) , ADR(a_tyXMLTableDataSnd[0].uiSize) , SIZEOF(a_tyXMLTableDataSnd[0]) , 30);

		ELSIF a_eMsgSend[0] = HermesMsgTypeNotification THEN
			fHermesFormNotification(ADR(a_tyXMLTableDataSnd) , p_tyDTStructure , tyNotificationSnd);
			fTableConvertToXML(ADR(sSnd) , ADR(udiSndMsgLen) , SIZEOF(sSnd) , ADR(a_tyXMLTableDataSnd) , ADR(a_tyXMLTableDataSnd[0].sTitle) , ADR(a_tyXMLTableDataSnd[0].sValue) , ADR(a_tyXMLTableDataSnd[0].uiSize) , SIZEOF(a_tyXMLTableDataSnd[0]) , 14);

		ELSIF a_eMsgSend[0] = HermesMsgTypeBoardAvailable THEN
			eStatus1	:= Error;
			udiStatus1	:= 10135;	//Board Available Request To Send From Upstream Hermes

		ELSIF a_eMsgSend[0] = HermesMsgTypeRevokeBoardAvl THEN
			eStatus1	:= Error;
			udiStatus1	:= 10136;	//Revoke Board Available Request To Send From Upstream Hermes

		ELSIF a_eMsgSend[0] = HermesMsgTypeMachineReady THEN
			fHermesFormMachineReady(ADR(a_tyXMLTableDataSnd) , p_tyDTStructure , tyMachineReady);
			fTableConvertToXML(ADR(sSnd) , ADR(udiSndMsgLen) , SIZEOF(sSnd) , ADR(a_tyXMLTableDataSnd) , ADR(a_tyXMLTableDataSnd[0].sTitle) , ADR(a_tyXMLTableDataSnd[0].sValue) , ADR(a_tyXMLTableDataSnd[0].uiSize) , SIZEOF(a_tyXMLTableDataSnd[0]) , 50);
			bReplyMcRdyId := FALSE;

		ELSIF a_eMsgSend[0] = HermesMsgTypeRevokeMachineReady THEN
			fHermesFormRevokeMachineReady(ADR(a_tyXMLTableDataSnd) , p_tyDTStructure);
			fTableConvertToXML(ADR(sSnd) , ADR(udiSndMsgLen) , SIZEOF(sSnd) , ADR(a_tyXMLTableDataSnd) , ADR(a_tyXMLTableDataSnd[0].sTitle) , ADR(a_tyXMLTableDataSnd[0].sValue) , ADR(a_tyXMLTableDataSnd[0].uiSize) , SIZEOF(a_tyXMLTableDataSnd[0]) , 8);

		ELSIF a_eMsgSend[0] = HermesMsgTypeStartTransport THEN
			fHermesFormStartTransport(ADR(a_tyXMLTableDataSnd) , p_tyDTStructure , tyStartTransport);
			fTableConvertToXML(ADR(sSnd) , ADR(udiSndMsgLen) , SIZEOF(sSnd) , ADR(a_tyXMLTableDataSnd) , ADR(a_tyXMLTableDataSnd[0].sTitle) , ADR(a_tyXMLTableDataSnd[0].sValue) , ADR(a_tyXMLTableDataSnd[0].uiSize) , SIZEOF(a_tyXMLTableDataSnd[0]) , 12);

		ELSIF a_eMsgSend[0] = HermesMsgTypeStopTransport THEN
			fHermesFormStopTransport(ADR(a_tyXMLTableDataSnd) , p_tyDTStructure , tyStopTransport);
			fTableConvertToXML(ADR(sSnd) , ADR(udiSndMsgLen) , SIZEOF(sSnd) , ADR(a_tyXMLTableDataSnd) , ADR(a_tyXMLTableDataSnd[0].sTitle) , ADR(a_tyXMLTableDataSnd[0].sValue) , ADR(a_tyXMLTableDataSnd[0].uiSize) , SIZEOF(a_tyXMLTableDataSnd[0]) , 12);

		ELSIF a_eMsgSend[0] = HermesMsgTypeTransportFinished THEN
			eStatus1	:= Error;
			udiStatus1	:= 10137;	//Transport Finished Request To Send From Upstream Hermes

		ELSIF a_eMsgSend[0] = HermesMsgTypeSetConfiguration THEN
			eStatus1	:= Error;
			udiStatus1	:= 10138;	//Set Configuration Request To Send From Upstream Hermes

		ELSIF a_eMsgSend[0] = HermesMsgTypeGetConfiguration THEN
			eStatus1	:= Error;
			udiStatus1	:= 10139;	//Get Configuration Request To Send From Upstream Hermes

		ELSIF a_eMsgSend[0] = HermesMsgTypeCurrConfiguration THEN
			eStatus1	:= Error;
			udiStatus1	:= 10140;	//Current Configuration Request To Send From Upstream Hermes

		ELSIF a_eMsgSend[0] = HermesMsgTypeBoardForecast THEN
			eStatus1	:= Error;
			udiStatus1	:= 10141;	//Board Forecast Request To Send From Upstream Hermes

		ELSIF a_eMsgSend[0] = HermesMsgTypeQueryBoardInfo THEN
			fHermesFormQueryBoardInfo(ADR(a_tyXMLTableDataSnd) , p_tyDTStructure , tyQueryBoardInfo);
			fTableConvertToXML(ADR(sSnd) , ADR(udiSndMsgLen) , SIZEOF(sSnd) , ADR(a_tyXMLTableDataSnd) , ADR(a_tyXMLTableDataSnd[0].sTitle) , ADR(a_tyXMLTableDataSnd[0].sValue) , ADR(a_tyXMLTableDataSnd[0].uiSize) , SIZEOF(a_tyXMLTableDataSnd[0]) , 12);
			//10142
		ELSIF a_eMsgSend[0] = HermesMsgTypeSendBoardInfo THEN
			eStatus1	:= Error;
			udiStatus1	:= 10159;	//Send Board Info Request To Send From Upstream Hermes

		ELSIF a_eMsgSend[0] = HermesMsgTypeQueryWorkOrderInfo THEN
			eStatus1	:= Error;
			udiStatus1	:= 10160;	//Query Work Order Info Request To Send From Upstream Hermes

		ELSIF a_eMsgSend[0] = HermesMsgTypeSendWorkOrderInfo THEN
			eStatus1	:= Error;
			udiStatus1	:= 10161;	//Send Work Order Info Request To Send From Upstream Hermes

		ELSIF a_eMsgSend[0] = HermesMsgTypeBoardArrived THEN
			eStatus1	:= Error;
			udiStatus1	:= 10162;	//BoardArrived Request To Send From Upstream Hermes

		ELSIF a_eMsgSend[0] = HermesMsgTypeBoardDeparted THEN
			eStatus1	:= Error;
			udiStatus1	:= 10163;	//BoardDeparted Request To Send From Upstream Hermes

		END_IF

		//Message Send
		IF p_bInternalUse = FALSE THEN
			fbSend.udiTCPIdent	:= udiTCPIdent;
			fbSend.udiSndSize	:= udiSndMsgLen;
			fbSend(bEn := TRUE);
		ELSE
			sInternalSnd	:= sSnd;
		END_IF

		IF (fbSend.udiStatus = 0) OR (p_bInternalUse = TRUE) THEN

			fLogDTConvert(ADR(sDT) , p_dtCurrDT);
			memset(ADR(a_sLogList[udiLogCntr]) , 0 , SIZEOF(a_sLogList[udiLogCntr]));
			memcpy(ADR(a_sLogList[udiLogCntr]) + LEN(a_sLogList[udiLogCntr]) , ADR(sDT) , LEN(sDT));
			memcpy(ADR(a_sLogList[udiLogCntr]) + LEN(a_sLogList[udiLogCntr]) , ADR('$r$n') , LEN('$r$n'));
			memcpy(ADR(a_sLogList[udiLogCntr]) + LEN(a_sLogList[udiLogCntr]) , ADR('SND_TO_US$r$n') , LEN('SND_TO_US$r$n'));
			memcpy(ADR(a_sLogList[udiLogCntr]) + LEN(a_sLogList[udiLogCntr]) , ADR(sSnd) , LEN(sSnd));
			memcpy(ADR(a_sLogList[udiLogCntr]) + LEN(a_sLogList[udiLogCntr]) , ADR('$r$n$r$n') , LEN('$r$n$r$n'));

			udiLogCntr	:= udiLogCntr + 1;
			IF udiLogCntr = 11 THEN
				udiLogCntr	:= 1;
			END_IF

			Act_Background_NotificationSnd;
			fHermesRmvOneMsgSend(ADR(a_eMsgSend) , ADR(udiMsgSendBffr));

			fbSend(bEn := FALSE);

		ELSIF (fbSend.udiStatus = 2321) AND (p_bInternalUse = FALSE) THEN
			bRstConnection	:= TRUE;

		ELSIF (fbSend.udiStatus < 65534) AND (p_bInternalUse = FALSE) THEN
			eStatus1	:= Error;

			IF fbSend.udiStatus = 2300 THEN
				udiStatus1	:= 10143;	//Invalid Ident While Sending Data
			ELSIF fbSend.udiStatus = 2320 THEN
				udiStatus1	:= 10144;	//TCP Retry Send Data Error While Sending Data
			ELSIF fbSend.udiStatus = 2322 THEN
				udiStatus1	:= 10145;	//TCP Send Data Error
			ELSE
				udiStatus1	:= fbSend.udiStatus;
			END_IF

		END_IF

	END_IF

END_ACTION
```

#### Act_Background_TCPClose.st - Do Not Change!!!
```iecst
(** 2021-08-01 **)
ACTION Act_Background_TCPClose:

	//Close TCP Connection
	IF p_bInternalUse = FALSE THEN
		fbClose.udiTCPIdent	:= udiTCPIdent;
		fbClose(bEn := TRUE);

		IF fbClose.udiStatus = 0 THEN
			udiTCPIdent	:= 0;
			fbClose(bEn := FALSE);

		ELSIF fbClose.udiStatus < 65534 THEN
			udiTCPIdent	:= 0;
			eStatus1	:= Error;

			IF fbClose.udiStatus = 2300 THEN
				udiStatus1	:= 10146;	//Invalid Ident While Closing TCP
			ELSIF fbClose.udiStatus = 2310 THEN
				udiStatus1	:= 10147;	//Closing TCP Error
			ELSE
				udiStatus1	:= fbClose.udiStatus;
			END_IF

		END_IF

	ELSE
		udiTCPIdent	:= 0;

	END_IF

END_ACTION
```

#### Act_Background_Stop.st - Do Not Change!!!
```iecst
(** 2021-08-01 **)
ACTION Act_Background_Stop:

	IF EDGEPOS(bStop) THEN

		fHermesAddOneMsgSend(ADR(a_eMsgSend) , ADR(udiMsgSendBffr) , HermesMsgTypeNotification);

		tyNotificationSnd.tyAvl.bSeverity			:= TRUE;
		tyNotificationSnd.tyAvl.bNotificationCode	:= TRUE;
		tyNotificationSnd.tyAvl.bDescription		:= TRUE;
		tyNotificationSnd.tyData.eSeverity			:= HermesSeverityInfo;
		tyNotificationSnd.tyData.iNotificationCode	:= 5;
		tyNotificationSnd.tyData.sDescription		:= 'Machine Shutdown';

	END_IF

	IF bStop = TRUE THEN

		IF a_eMsgSend[0] = HermesMsgTypeNA THEN

			bRstConnection	:= TRUE;

			IF udiTCPIdent = 0 THEN

				bRun	:= FALSE;

			END_IF

		END_IF

	END_IF

END_ACTION
```

#### Act_Background_Log.st - Do Not Change!!!
```iecst
(** 2021-08-01 **)
ACTION Act_Background_Log:

	IF eStatus3 <> Error THEN

		IF udiWriteLogCntr <> udiLogCntr THEN

			CASE iWriteLogStep OF

				0:
					dtCurrDTTemp			:= p_dtCurrDT;
					fbFileAppend1.sFile		:= DT_TO_STRING(dtCurrDTTemp);
					fbFileAppend1.sFile		:= MID(fbFileAppend1.sFile , 10 , 4);
					fbFileAppend1.sFile		:= CONCAT('_' , fbFileAppend1.sFile);
					fbFileAppend1.sFile		:= CONCAT(p_sProgNm , fbFileAppend1.sFile);
					fbFileAppend1.sFile		:= CONCAT(fbFileAppend1.sFile , '.dat');

					fbFileAppend1.p_Src		:= ADR(a_sLogList[udiWriteLogCntr]);
					fbFileAppend1.udiLen	:= LEN(a_sLogList[udiWriteLogCntr]);

					iWriteLogStep	:= 1;

				1:
					fbFileAppend1(bEn := TRUE);
					IF fbFileAppend1.udiStatus = 0 THEN
						fbFileAppend1(bEn := FALSE);

						udiWriteLogCntr	:= udiWriteLogCntr + 1;
						IF udiWriteLogCntr = 11 THEN
							udiWriteLogCntr	:= 1;
						END_IF

						iWriteLogStep	:= 0;

					ELSIF fbFileAppend1.udiStatus < 65534 THEN
						eStatus3	:= Error;

						IF fbFileAppend1.udiStatus = 1900 THEN
							udiStatus3	:= 10148;	//File Open Error While Writing Log
						ELSIF fbFileAppend1.udiStatus = 1901 THEN
							udiStatus3	:= 10149;	//File Create Error While Writing Log
						ELSIF fbFileAppend1.udiStatus = 1913 THEN
							udiStatus3	:= 10150;	//Get File Info Error While Writing Log
						ELSIF fbFileAppend1.udiStatus = 1903 THEN
							udiStatus3	:= 10151;	//File Write Error While Writing Log
						ELSIF fbFileAppend1.udiStatus = 1904 THEN
							udiStatus3	:= 10152;	//File Close Error While Writing Log
						ELSIF fbFileAppend1.udiStatus = 1914 THEN
							udiStatus3	:= 10153;	//Directory Does Not Exist While Writing Log
						ELSE
							udiStatus3	:= fbFileAppend1.udiStatus;
						END_IF

						iWriteLogStep	:= 0;

					END_IF

			END_CASE

		END_IF

	END_IF

END_ACTION
```

#### Act_Background_AccData.st - Change By Project
```iecst
(** 2021-08-01 **)
ACTION Act_Background_AccData: //Accept BoardAvailable Data from Upstream

	CASE usiAccDataStep OF
		0:
			//Request Accept Data
			IF bUSRdy = TRUE AND eMainStatus <> Error AND bAccDataReq = TRUE THEN
				usiAccDataStep	:= 1;
			END_IF
			//bUSRdy := fbSequenceUS.bUSRdy;
			//bUSRdy:= (eState = HermesStateBoardAvailable) OR (eState = HermesStateAvailableAndReady) OR (eState >= HermesStateTransporting);
		1:
			//Manual Accept Data Check
			IF bAccDataReq = TRUE THEN
				IF p_bMcParamMnlAccData = TRUE THEN
					bAccDataMnl	:= TRUE;

					tyInfoData.sProgNm		:= p_sProgNm;
					tyInfoData.udiCode		:= 10000;
					tyInfoData.eSeverity	:= AlmSeverityInfo;
					tyInfoData.sAlmMsg		:= p_sInfoMsg;

					IF p_bUIAccData = TRUE THEN
						p_bUIAccData    := FALSE; //2023_07_26_Debug for Manual Accept Data automatically accept after product change many times
						bAccDataMnl		:= FALSE;
						usiAccDataStep	:= 2;
					END_IF
				ELSE
					bAccDataMnl		:= FALSE;
					p_bUIAccData    := FALSE; //2023_07_26_Debug for Manual Accept Data automatically accept after product change many times
					usiAccDataStep	:= 2;
				END_IF
			ELSE
				bAccDataMnl		:= FALSE;
				usiAccDataStep	:= 4;
			END_IF

		2:
			IF bAccDataReq = TRUE  THEN
				IF p_bAccNewRcpCond = TRUE THEN //In Auto Mode, and empty
					usiAccDataStep	:= 3;
					IF p_bNtParamAutoRcpPrep AND NOT(p_bMcParamAutoRcpDis) THEN
						CASE p_eNtParamAutoRcpPrecededBy OF
							PrecededBySelf:
								usiAccDataStep	:= 4;
							PrecededByF1:
								usiAccDataStep	:= 3;
						END_CASE
					END_IF
				ELSE
					//Info Message
					tyInfoData.sProgNm		:= p_sProgNm;
					tyInfoData.udiCode		:= 10000;
					tyInfoData.eSeverity	:= AlmSeverityInfo;
					tyInfoData.sAlmMsg		:= p_sInfoMsg;
				END_IF
			ELSE
				usiAccDataStep	:= 4;
			END_IF

		3:
			//Sync Recipe
			IF bOverWriteWidth = TRUE OR bOverWriteSlt = TRUE THEN

				//Accept New Recipe Width
				IF bOverWriteWidth = TRUE THEN
					p_tyProdRcpCurrRcp.diWidthInUM	:= diReqWidthInUM;
				END_IF

				//Accept New Recipe Slot
				IF bOverWriteSlt = TRUE THEN
					p_tyProdRcpCurrRcp.diMaxSltValue := diReqMaxSltValue;
					p_tyProdRcpCurrRcp.diMinSltValue := diReqMinSltValue;
					p_tyProdRcpCurrRcp.diPitch := diReqPitch;
				END_IF

			ELSE

				//Accept New Recipe Name
				FOR i := 1 TO 2000 DO
					IF sReqRecipeNm = pa_tyProdRcpList[i].sRcpNm THEN
						p_tyProdRcpCurrRcp	:= pa_tyProdRcpList[i];
						EXIT;
					END_IF
				END_FOR

				IF i > 2000 THEN
					//Recipe Not Exist
					eStatus4	:= Error;
					udiStatus4	:= 10169;	//New Recipe Not Found In Product Recipe List

					fHermesAddOneMsgSend(ADR(a_eMsgSend) , ADR(udiMsgSendBffr) , HermesMsgTypeNotification);

					tyNotificationSnd.tyAvl.bSeverity			:= TRUE;
					tyNotificationSnd.tyAvl.bNotificationCode	:= TRUE;
					tyNotificationSnd.tyAvl.bDescription		:= TRUE;
					tyNotificationSnd.tyData.eSeverity			:= HermesSeverityError;
					tyNotificationSnd.tyData.iNotificationCode	:= UDINT_TO_INT(udiStatus4);
					tyNotificationSnd.tyData.sDescription		:= a_tyAlmText[udiStatus4].sAlmText;

				END_IF

			END_IF

			usiAccDataStep	:= 4;

		4:
			//Clear Info Message
			tyInfoData.sProgNm		:= '';
			tyInfoData.udiCode		:= 0;
			tyInfoData.eSeverity	:= AlmSeverityNA;
			tyInfoData.sAlmMsg		:= '';

			usiAccDataStep	:= 0;

	END_CASE

END_ACTION
```

#### Act_Background_BFAccData.st - Change By Project
```iecst
(** 2021-08-01 **)
ACTION Act_Background_BFAccData: //Accept BoardForecast Data from Upstream

	CASE usiBFAccDataStep OF
		0:
			//Request Accept Data
			IF bProcessBoardForecastId = TRUE AND eMainStatus <> Error AND bBFAccDataReq = TRUE THEN
				usiBFAccDataStep	:= 1;
			END_IF

		1:
			//Manual Accept Data Check
			IF bBFAccDataReq = TRUE THEN
				IF p_bMcParamMnlAccData = TRUE THEN
					bAccDataMnl	:= TRUE; //use bAccDataMnl instead of bBFAccDataMnl

					tyInfoData.sProgNm		:= p_sProgNm;
					tyInfoData.udiCode		:= 10000;
					tyInfoData.eSeverity	:= AlmSeverityInfo;
					tyInfoData.sAlmMsg		:= p_sInfoMsg;

					IF p_bUIAccData = TRUE THEN
						bAccDataMnl		:= FALSE;
						usiBFAccDataStep	:= 2;
					END_IF
				ELSE
					bAccDataMnl		:= FALSE;
					usiBFAccDataStep	:= 2;
				END_IF
			ELSE
				bAccDataMnl		:= FALSE;
				usiBFAccDataStep	:= 4;
			END_IF

		2:
			IF bBFAccDataReq = TRUE THEN
				IF p_bAccNewRcpCond = TRUE THEN //In Auto Mode, and empty
					usiBFAccDataStep	:= 3;
					IF p_bNtParamAutoRcpPrep AND NOT(p_bMcParamAutoRcpDis) THEN
						CASE p_eNtParamAutoRcpPrecededBy OF
							PrecededBySelf:
								usiBFAccDataStep	:= 4;
							PrecededByF1:
								usiBFAccDataStep	:= 3;
						END_CASE
					END_IF
				ELSE
					//Info Message
					tyInfoData.sProgNm		:= p_sProgNm;
					tyInfoData.udiCode		:= 10000;
					tyInfoData.eSeverity	:= AlmSeverityInfo;
					tyInfoData.sAlmMsg		:= p_sInfoMsg;
				END_IF
			ELSE
				usiBFAccDataStep	:= 4;
			END_IF

		3:
			//Sync Recipe
			IF bBFOverWriteWidth = TRUE OR bBFOverWriteSlt = TRUE THEN

				//Accept New Recipe Width
				IF bBFOverWriteWidth = TRUE THEN
					p_tyProdRcpCurrRcp.diWidthInUM	:= diReqWidthInUM;
				END_IF

				//Accept New Recipe Slot
				IF bBFOverWriteSlt = TRUE THEN
					diReqMaxSltValue;
					diReqMinSltValue;
					diReqPitch;
				END_IF

			ELSE

				//Accept New Recipe Name
				FOR i := 1 TO 2000 DO
					IF sReqRecipeNm = pa_tyProdRcpList[i].sRcpNm THEN
						p_tyProdRcpCurrRcp	:= pa_tyProdRcpList[i];
						EXIT;
					END_IF
				END_FOR

				IF i > 2000 THEN
					//Recipe Not Exist
					eStatus4	:= Error;
					udiStatus4	:= 10169;	//New Recipe Not Found In Product Recipe List

					fHermesAddOneMsgSend(ADR(a_eMsgSend) , ADR(udiMsgSendBffr) , HermesMsgTypeNotification);

					tyNotificationSnd.tyAvl.bSeverity			:= TRUE;
					tyNotificationSnd.tyAvl.bNotificationCode	:= TRUE;
					tyNotificationSnd.tyAvl.bDescription		:= TRUE;
					tyNotificationSnd.tyData.eSeverity			:= HermesSeverityError;
					tyNotificationSnd.tyData.iNotificationCode	:= 6; //BoreForecast Error
					tyNotificationSnd.tyData.sDescription		:= a_tyAlmText[udiStatus4].sAlmText;

				END_IF

			END_IF

			usiBFAccDataStep	:= 4;

		4:
			//Clear Info Message
			tyInfoData.sProgNm		:= '';
			tyInfoData.udiCode		:= 0;
			tyInfoData.eSeverity	:= AlmSeverityNA;
			tyInfoData.sAlmMsg		:= '';
			usiBFAccDataStep	:= 0;
			bReplyMcRdyId           := TRUE; //add
			bProcessBoardForecastId := FALSE; //add
	END_CASE

END_ACTION
```

#### Act_CombineErr.st - Do Not Change!!!
```iecst
(** 2021-08-01 **)
ACTION Act_CombineErr:

	//Combine Error
	IF eStatus = Error OR eStatus1 = Error OR eStatus2 = Error OR eStatus3 = Error OR eStatus4 = Error THEN
		eMainStatus	:= Error;
	ELSE
		eMainStatus	:= eStatus;
	END_IF

END_ACTION
```

#### Act_Alarm.st - Do Not Change!!!
```iecst
(** 2019-03-25 **)
ACTION Act_Alarm:

	//Error
	IF EDGEPOS(eStatus = Error) THEN

		tyAlmData.sProgNm		:= p_sProgNm;
		tyAlmData.udiCode		:= udiStatus;
		tyAlmData.eSeverity		:= AlmSeverityError;
		tyAlmData.udiRunTime	:= tyAlmData.udiRunTime + 1;
		tyAlmData.bAlm			:= TRUE;
		tyAlmData.udiModuleNum  := udiModuleNum;
		g_sUSHermesAProgNm		:= p_sProgNm;

		//Get Error Message
		IF tyAlmData.udiCode < 10000 OR tyAlmData.udiCode > 10199 THEN
			tyAlmData.sAlmMsg	:= 'Unknown';
			tyAlmData.sRcyMsg	:= 'Unknown';
		ELSE
			tyAlmData.sAlmMsg	:= a_tyAlmText[tyAlmData.udiCode].sAlmText;
			tyAlmData.sRcyMsg	:= a_tyAlmText[tyAlmData.udiCode].sRcyText;
		END_IF

		sStatTxt	:= tyAlmData.sAlmMsg;

	ELSIF bRstErr AND (tyAlmData.udiCode <> 0) THEN

		tyAlmData.udiCode	:= 0;
		tyAlmData.eSeverity	:= AlmSeverityNA;
		tyAlmData.sAlmMsg	:= '';
		tyAlmData.sRcyMsg	:= '';
		tyAlmData.bAlm			:= FALSE;
		sStatTxt	:= a_sStatText[eStat];

	END_IF

END_ACTION
```
